C05442=1098.979,27.951,-55.035,176.233,15.027,151.969
C05443=1098.973,27.702,-55.021,176.230,15.027,151.970
C05444=1098.967,27.452,-55.005,176.228,15.026,151.970
C05445=1098.962,27.202,-54.991,176.226,15.025,151.971
C05446=1098.956,26.952,-54.976,176.224,15.025,151.971
C05447=1098.951,26.703,-54.961,176.221,15.024,151.971
C05448=1098.944,26.454,-54.946,176.219,15.023,151.972
C05449=1098.939,26.204,-54.931,176.217,15.022,151.972
C05450=1098.933,25.955,-54.916,176.215,15.022,151.972
C05451=1098.927,25.705,-54.902,176.212,15.021,151.973
C05452=1098.922,25.455,-54.887,176.210,15.020,151.973
C05453=1098.916,25.206,-54.872,176.208,15.020,151.973
C05454=1098.910,24.957,-54.857,176.206,15.019,151.974
C05455=1098.904,24.708,-54.843,176.203,15.018,151.974
C05456=1098.899,24.458,-54.828,176.201,15.018,151.974
C05457=1098.893,24.208,-54.813,176.199,15.017,151.975
C05458=1098.887,23.959,-54.799,176.197,15.016,151.975
C05459=1098.881,23.709,-54.783,176.194,15.015,151.975
C05460=1098.876,23.460,-54.769,176.192,15.015,151.976
C05461=1098.869,23.210,-54.754,176.190,15.014,151.976
C05462=1098.863,22.961,-54.740,176.188,15.013,151.976
C05463=1098.858,22.712,-54.724,176.186,15.012,151.976
C05464=1098.852,22.461,-54.710,176.183,15.012,151.977
C05465=1098.847,22.213,-54.696,176.182,15.011,151.977
C05466=1098.841,21.963,-54.680,176.180,15.010,151.977
C05467=1098.835,21.713,-54.666,176.177,15.009,151.978
C05468=1098.830,21.464,-54.652,176.175,15.009,151.978
C05469=1098.823,21.214,-54.637,176.173,15.008,151.979
C05470=1098.819,20.964,-54.622,176.171,15.008,151.979
C05471=1098.813,20.716,-54.608,176.168,15.006,151.979
C05472=1098.806,20.466,-54.593,176.166,15.006,151.979
C05473=1098.801,20.216,-54.579,176.164,15.005,151.980
C05474=1098.795,19.967,-54.564,176.162,15.005,151.980
C05475=1098.789,19.717,-54.549,176.159,15.004,151.980
C05476=1098.784,19.468,-54.535,176.157,15.003,151.981
C05477=1098.778,19.218,-54.520,176.155,15.002,151.981
C05478=1098.772,18.969,-54.505,176.153,15.002,151.981
C05479=1098.766,18.719,-54.491,176.151,15.001,151.982
C05480=1098.760,18.470,-54.477,176.149,15.000,151.982
C05481=1098.755,18.220,-54.462,176.147,14.999,151.982
C05482=1098.749,17.970,-54.447,176.145,14.999,151.983
C05483=1098.743,17.721,-54.433,176.143,14.998,151.983
C05484=1098.738,17.472,-54.419,176.140,14.997,151.983
C05485=1098.731,17.222,-54.404,176.138,14.996,151.984
C05486=1098.726,16.973,-54.390,176.136,14.996,151.984
C05487=1098.720,16.724,-54.375,176.134,14.995,151.984
C05488=1098.714,16.473,-54.361,176.131,14.994,151.985
C05489=1098.709,16.224,-54.346,176.129,14.993,151.985
C05490=1098.702,15.952,-54.331,176.127,14.993,151.985
C05491=1098.696,15.680,-54.315,176.125,14.992,151.985
C05492=1098.690,15.408,-54.300,176.123,14.991,151.986
C05493=1098.684,15.136,-54.284,176.120,14.991,151.986
C05494=1098.678,14.886,-54.269,176.118,14.989,151.986
C05495=1098.672,14.637,-54.255,176.116,14.988,151.987
C05496=1098.666,14.388,-54.241,176.114,14.988,151.987
C05497=1098.660,14.137,-54.227,176.112,14.987,151.987
C05498=1098.655,13.889,-54.212,176.109,14.986,151.988
C05499=1098.649,13.639,-54.198,176.107,14.985,151.988
C05500=1098.643,13.389,-54.183,176.105,14.985,151.988
C05501=1098.637,13.140,-54.169,176.103,14.984,151.989
C05502=1098.631,12.891,-54.155,176.101,14.984,151.989
C05503=1098.625,12.640,-54.140,176.098,14.983,151.989
C05504=1098.620,12.391,-54.127,176.097,14.982,151.990
C05505=1098.614,12.142,-54.112,176.095,14.981,151.990
C05506=1098.608,11.892,-54.098,176.092,14.981,151.990
C05507=1098.602,11.642,-54.085,176.091,14.980,151.990
C05508=1098.596,11.393,-54.070,176.088,14.979,151.991
C05509=1098.590,11.143,-54.056,176.086,14.978,151.991
C05510=1098.584,10.894,-54.041,176.084,14.978,151.991
C05511=1098.579,10.645,-54.027,176.082,14.977,151.992
C05512=1098.573,10.394,-54.013,176.080,14.976,151.992
C05513=1098.567,10.145,-53.998,176.077,14.975,151.992
C05514=1098.561,9.896,-53.985,176.075,14.975,151.993
C05515=1098.556,9.646,-53.971,176.073,14.974,151.993
C05516=1098.550,9.397,-53.956,176.072,14.973,151.993
C05517=1098.543,9.147,-53.943,176.070,14.972,151.993
C05518=1098.538,8.898,-53.929,176.067,14.972,151.994
C05519=1098.532,8.648,-53.915,176.065,14.971,151.994
C05520=1098.526,8.399,-53.900,176.063,14.970,151.994
C05521=1098.520,8.149,-53.886,176.061,14.969,151.995
C05522=1098.515,7.899,-53.872,176.059,14.969,151.995
C05523=1098.510,7.650,-53.858,176.056,14.968,151.995
C05524=1098.502,7.400,-53.844,176.054,14.967,151.996
C05525=1098.497,7.151,-53.830,176.052,14.966,151.996
C05526=1098.491,6.901,-53.816,176.051,14.965,151.996
C05527=1098.486,6.652,-53.802,176.048,14.965,151.997
C05528=1098.480,6.402,-53.787,176.046,14.964,151.997
C05529=1098.474,6.153,-53.773,176.044,14.963,151.997
C05530=1098.469,5.903,-53.760,176.042,14.962,151.997
C05531=1098.462,5.654,-53.746,176.040,14.962,151.998
C05532=1098.457,5.404,-53.732,176.038,14.961,151.998
C05533=1098.451,5.154,-53.718,176.036,14.961,151.998
C05534=1098.445,4.905,-53.704,176.033,14.959,151.999
C05535=1098.440,4.655,-53.690,176.031,14.958,151.999
C05536=1098.433,4.406,-53.677,176.030,14.958,151.999
C05537=1098.428,4.156,-53.663,176.028,14.957,151.999
C05538=1098.422,3.907,-53.649,176.026,14.956,152.000
C05539=1098.416,3.657,-53.635,176.023,14.955,152.000
C05540=1098.411,3.408,-53.620,176.021,14.955,152.000
C05541=1098.404,3.158,-53.607,176.019,14.954,152.001
C05542=1098.399,2.909,-53.593,176.017,14.953,152.001
C05543=1098.393,2.659,-53.579,176.015,14.952,152.001
C05544=1098.388,2.410,-53.565,176.014,14.952,152.001
C05545=1098.382,2.160,-53.551,176.011,14.950,152.002
C05546=1098.376,1.910,-53.538,176.009,14.950,152.002
C05547=1098.370,1.661,-53.524,176.007,14.949,152.002
C05548=1098.365,1.411,-53.510,176.005,14.949,152.003
C05549=1098.359,1.161,-53.496,176.003,14.948,152.003
C05550=1098.353,0.912,-53.483,176.001,14.947,152.003
C05551=1098.348,0.663,-53.469,175.998,14.946,152.003
C05552=1098.342,0.413,-53.455,175.997,14.945,152.004
C05553=1098.337,0.163,-53.441,175.995,14.944,152.004
C05554=1098.330,-0.107,-53.426,175.993,14.943,152.004
C05555=1098.324,-0.377,-53.412,175.990,14.942,152.004
C05556=1098.317,-0.646,-53.396,175.988,14.941,152.005
C05557=1098.311,-0.917,-53.381,175.986,14.941,152.005
C05558=1098.305,-1.166,-53.368,175.983,14.940,152.005
C05559=1098.300,-1.416,-53.354,175.982,14.939,152.006
C05560=1098.294,-1.665,-53.340,175.980,14.938,152.006
C05561=1098.289,-1.915,-53.327,175.978,14.938,152.006
C05562=1098.283,-2.165,-53.314,175.976,14.937,152.006
C05563=1098.277,-2.414,-53.300,175.974,14.936,152.007
C05564=1098.272,-2.664,-53.286,175.971,14.935,152.007
C05565=1098.265,-2.913,-53.273,175.970,14.934,152.007
C05566=1098.260,-3.163,-53.259,175.968,14.933,152.007
C05567=1098.255,-3.412,-53.245,175.966,14.932,152.008
C05568=1098.248,-3.661,-53.232,175.964,14.932,152.008
C05569=1098.242,-3.912,-53.218,175.962,14.931,152.008
C05570=1098.236,-4.161,-53.204,175.960,14.930,152.008
C05571=1098.231,-4.411,-53.190,175.957,14.929,152.009
C05572=1098.225,-4.660,-53.178,175.955,14.929,152.009
C05573=1098.219,-4.910,-53.164,175.953,14.928,152.009
C05574=1098.213,-5.159,-53.151,175.952,14.927,152.010
C05575=1098.207,-5.409,-53.137,175.950,14.926,152.010
C05576=1098.201,-5.658,-53.124,175.948,14.926,152.010
C05577=1098.196,-5.908,-53.110,175.946,14.925,152.010
C05578=1098.190,-6.157,-53.096,175.943,14.924,152.011
C05579=1098.184,-6.408,-53.083,175.941,14.923,152.011
C05580=1098.178,-6.657,-53.070,175.940,14.922,152.011
C05581=1098.172,-6.907,-53.056,175.938,14.921,152.012
C05582=1098.166,-7.156,-53.042,175.935,14.921,152.012
C05583=1098.160,-7.406,-53.029,175.934,14.920,152.012
C05584=1098.155,-7.655,-53.016,175.932,14.920,152.013
C05585=1098.149,-7.905,-53.002,175.930,14.919,152.013
C05586=1098.143,-8.154,-52.989,175.927,14.917,152.013
C05587=1098.137,-8.404,-52.975,175.925,14.917,152.013
C05588=1098.131,-8.653,-52.962,175.923,14.916,152.014
C05589=1098.126,-8.903,-52.949,175.922,14.915,152.014
C05590=1098.120,-9.153,-52.935,175.920,14.915,152.014
C05591=1098.114,-9.402,-52.922,175.918,14.914,152.014
C05592=1098.108,-9.652,-52.909,175.916,14.913,152.015
C05593=1098.102,-9.901,-52.896,175.914,14.912,152.015
C05594=1098.097,-10.151,-52.882,175.911,14.911,152.015
C05595=1098.090,-10.400,-52.869,175.909,14.910,152.015
C05596=1098.085,-10.650,-52.855,175.908,14.909,152.016
C05597=1098.079,-10.900,-52.842,175.906,14.909,152.016
C05598=1098.074,-11.149,-52.828,175.904,14.908,152.016
C05599=1098.068,-11.399,-52.816,175.902,14.907,152.016
C05600=1098.061,-11.648,-52.802,175.900,14.906,152.017
C05601=1098.056,-11.898,-52.789,175.898,14.906,152.017
C05602=1098.050,-12.148,-52.776,175.896,14.904,152.017
C05603=1098.045,-12.397,-52.762,175.894,14.904,152.018
C05604=1098.038,-12.647,-52.749,175.892,14.903,152.018
C05605=1098.033,-12.896,-52.736,175.890,14.902,152.018
C05606=1098.027,-13.146,-52.722,175.888,14.901,152.018
C05607=1098.021,-13.396,-52.710,175.886,14.901,152.019
C05608=1098.016,-13.645,-52.696,175.884,14.900,152.019
C05609=1098.009,-13.895,-52.683,175.882,14.899,152.019
C05610=1098.004,-14.144,-52.671,175.881,14.898,152.019
C05611=1097.999,-14.393,-52.657,175.878,14.897,152.020
C05612=1097.993,-14.643,-52.644,175.876,14.896,152.020
C05613=1097.987,-14.893,-52.631,175.874,14.896,152.020
C05614=1097.981,-15.143,-52.618,175.872,14.895,152.020
C05615=1097.975,-15.392,-52.605,175.870,14.894,152.021
C05616=1097.969,-15.641,-52.591,175.868,14.893,152.021
C05617=1097.963,-15.891,-52.579,175.867,14.893,152.021
C05618=1097.957,-16.160,-52.564,175.865,14.892,152.021
C05619=1097.950,-16.428,-52.551,175.862,14.891,152.022
C05620=1097.944,-16.697,-52.536,175.860,14.890,152.022
C05621=1097.938,-16.965,-52.523,175.858,14.890,152.022
C05622=1097.932,-17.214,-52.509,175.856,14.889,152.023
C05623=1097.927,-17.465,-52.496,175.854,14.888,152.023
C05624=1097.920,-17.714,-52.483,175.852,14.887,152.023
C05625=1097.914,-17.964,-52.470,175.850,14.886,152.023
C05626=1097.908,-18.213,-52.457,175.848,14.885,152.024
C05627=1097.902,-18.463,-52.444,175.846,14.885,152.024
C05628=1097.897,-18.712,-52.431,175.844,14.884,152.024
C05629=1097.892,-18.962,-52.418,175.842,14.883,152.025
C05630=1097.885,-19.211,-52.405,175.840,14.882,152.025
C05631=1097.879,-19.461,-52.393,175.838,14.882,152.025
C05632=1097.873,-19.710,-52.379,175.837,14.881,152.025
C05633=1097.867,-19.960,-52.367,175.835,14.880,152.026
C05634=1097.862,-20.210,-52.354,175.833,14.879,152.026
C05635=1097.856,-20.459,-52.340,175.831,14.879,152.026
C05636=1097.850,-20.709,-52.328,175.829,14.878,152.026
C05637=1097.844,-20.959,-52.315,175.827,14.877,152.026
C05638=1097.839,-21.208,-52.302,175.825,14.875,152.027
C05639=1097.833,-21.458,-52.290,175.823,14.875,152.027
C05640=1097.827,-21.707,-52.276,175.821,14.874,152.027
C05641=1097.821,-21.957,-52.263,175.819,14.873,152.027
C05642=1097.815,-22.206,-52.250,175.817,14.872,152.028
C05643=1097.809,-22.456,-52.238,175.815,14.872,152.028
C05644=1097.803,-22.706,-52.225,175.814,14.871,152.028
C05645=1097.798,-22.955,-52.212,175.812,14.870,152.029
C05646=1097.792,-23.205,-52.200,175.810,14.869,152.029
C05647=1097.786,-23.455,-52.187,175.808,14.869,152.029
C05648=1097.780,-23.704,-52.173,175.806,14.868,152.029
C05649=1097.774,-23.954,-52.161,175.804,14.867,152.030
C05650=1097.768,-24.204,-52.148,175.802,14.866,152.030
C05651=1097.763,-24.453,-52.136,175.800,14.866,152.030
C05652=1097.757,-24.702,-52.123,175.798,14.864,152.030
C05653=1097.751,-24.952,-52.110,175.796,14.864,152.031
C05654=1097.745,-25.202,-52.097,175.794,14.863,152.031
C05655=1097.739,-25.451,-52.084,175.792,14.862,152.031
C05656=1097.734,-25.701,-52.072,175.790,14.861,152.031
C05657=1097.728,-25.951,-52.059,175.789,14.860,152.032
C05658=1097.723,-26.201,-52.046,175.787,14.859,152.032
C05659=1097.717,-26.450,-52.034,175.785,14.859,152.032
C05660=1097.710,-26.700,-52.020,175.783,14.858,152.032
C05661=1097.705,-26.949,-52.008,175.781,14.857,152.033
C05662=1097.699,-27.199,-51.996,175.779,14.857,152.033
C05663=1097.693,-27.449,-51.983,175.777,14.856,152.033
C05664=1097.687,-27.698,-51.970,175.776,14.855,152.033
C05665=1097.681,-27.948,-51.957,175.774,14.854,152.034
C05666=1097.676,-28.197,-51.945,175.772,14.854,152.034
C05667=1097.669,-28.447,-51.933,175.770,14.853,152.034
C05668=1097.663,-28.696,-51.921,175.768,14.852,152.034
C05669=1097.657,-28.946,-51.907,175.766,14.851,152.035
C05670=1097.651,-29.196,-51.895,175.764,14.851,152.035
C05671=1097.646,-29.445,-51.883,175.762,14.850,152.035
C05672=1097.640,-29.695,-51.870,175.760,14.849,152.035
C05673=1097.634,-29.945,-51.858,175.759,14.848,152.036
C05674=1097.628,-30.194,-51.845,175.757,14.848,152.036
C05675=1097.622,-30.444,-51.832,175.754,14.846,152.036
C05676=1097.617,-30.693,-51.819,175.752,14.846,152.036
C05677=1097.611,-30.943,-51.807,175.750,14.845,152.037
C05678=1097.604,-31.192,-51.795,175.748,14.844,152.037
C05679=1097.598,-31.442,-51.782,175.747,14.843,152.037
C05680=1097.593,-31.691,-51.770,175.745,14.842,152.037
C05681=1097.587,-31.941,-51.758,175.743,14.841,152.038
C05682=1097.581,-32.209,-51.744,175.741,14.841,152.038
C05683=1097.575,-32.477,-51.731,175.739,14.840,152.038
C05684=1097.567,-32.744,-51.717,175.737,14.839,152.038
C05685=1097.561,-33.012,-51.704,175.736,14.839,152.039
C05686=1097.556,-33.261,-51.692,175.734,14.838,152.039
C05687=1097.550,-33.511,-51.680,175.732,14.837,152.039
C05688=1097.544,-33.761,-51.667,175.730,14.836,152.039
C05689=1097.538,-34.010,-51.654,175.728,14.836,152.040
C05690=1097.532,-34.259,-51.642,175.726,14.835,152.040
C05691=1097.526,-34.509,-51.630,175.724,14.834,152.040
C05692=1097.520,-34.759,-51.617,175.722,14.833,152.040
C05693=1097.515,-35.008,-51.605,175.721,14.833,152.041
C05694=1097.509,-35.258,-51.592,175.719,14.832,152.041
C05695=1097.503,-35.508,-51.580,175.717,14.831,152.041
C05696=1097.497,-35.758,-51.569,175.715,14.830,152.042
C05697=1097.492,-36.007,-51.556,175.713,14.830,152.042
C05698=1097.486,-36.257,-51.544,175.711,14.829,152.042
C05699=1097.480,-36.507,-51.531,175.709,14.827,152.042
C05700=1097.474,-36.756,-51.519,175.707,14.826,152.042
C05701=1097.468,-37.006,-51.507,175.705,14.826,152.043
C05702=1097.462,-37.256,-51.495,175.703,14.825,152.043
C05703=1097.457,-37.505,-51.482,175.701,14.824,152.043
C05704=1097.451,-37.755,-51.470,175.699,14.823,152.044
C05705=1097.445,-38.005,-51.457,175.698,14.823,152.044
C05706=1097.439,-38.254,-51.445,175.696,14.822,152.044
C05707=1097.433,-38.503,-51.433,175.695,14.822,152.044
C05708=1097.427,-38.753,-51.421,175.693,14.821,152.044
C05709=1097.422,-39.003,-51.408,175.691,14.820,152.045
C05710=1097.415,-39.253,-51.397,175.689,14.819,152.045
C05711=1097.409,-39.503,-51.385,175.687,14.818,152.045
C05712=1097.404,-39.752,-51.372,175.685,14.818,152.045
C05713=1097.397,-40.001,-51.360,175.684,14.817,152.046
C05714=1097.391,-40.251,-51.348,175.682,14.816,152.046
C05715=1097.386,-40.500,-51.336,175.680,14.816,152.046
C05716=1097.379,-40.750,-51.324,175.678,14.815,152.046
C05717=1097.374,-41.000,-51.312,175.676,14.814,152.047
C05718=1097.369,-41.250,-51.300,175.674,14.813,152.047
C05719=1097.362,-41.499,-51.288,175.672,14.813,152.047
C05720=1097.356,-41.749,-51.275,175.670,14.812,152.047
C05721=1097.350,-41.998,-51.264,175.669,14.811,152.048
C05722=1097.344,-42.248,-51.251,175.667,14.810,152.048
C05723=1097.338,-42.498,-51.239,175.665,14.810,152.048
C05724=1097.332,-42.747,-51.228,175.663,14.809,152.049
C05725=1097.326,-42.997,-51.215,175.661,14.808,152.049
C05726=1097.321,-43.247,-51.203,175.659,14.807,152.049
C05727=1097.315,-43.497,-51.192,175.657,14.807,152.049
C05728=1097.309,-43.746,-51.179,175.656,14.806,152.049
C05729=1097.303,-43.995,-51.168,175.654,14.805,152.050
C05730=1097.297,-44.245,-51.155,175.652,14.804,152.050
C05731=1097.291,-44.496,-51.143,175.650,14.803,152.050
C05732=1097.285,-44.745,-51.132,175.648,14.803,152.050
C05733=1097.279,-44.994,-51.119,175.646,14.802,152.051
C05734=1097.273,-45.243,-51.107,175.644,14.801,152.051
C05735=1097.268,-45.494,-51.096,175.643,14.800,152.051
C05736=1097.261,-45.743,-51.084,175.641,14.800,152.052
C05737=1097.256,-45.993,-51.071,175.639,14.799,152.052
C05738=1097.250,-46.243,-51.060,175.637,14.798,152.052
C05739=1097.244,-46.492,-51.048,175.635,14.797,152.052
C05740=1097.238,-46.742,-51.035,175.634,14.797,152.053
C05741=1097.232,-46.992,-51.024,175.632,14.797,152.053
C05742=1097.227,-47.241,-51.012,175.630,14.795,152.053
C05743=1097.220,-47.491,-51.000,175.629,14.795,152.053
C05744=1097.215,-47.741,-50.989,175.627,14.794,152.053
C05745=1097.208,-47.990,-50.977,175.625,14.793,152.054
C05746=1097.202,-48.258,-50.964,175.623,14.792,152.054
C05747=1097.196,-48.526,-50.951,175.621,14.792,152.054
C05748=1097.190,-48.794,-50.938,175.619,14.791,152.054
C05749=1097.183,-49.061,-50.926,175.616,14.790,152.055
C05750=1097.178,-49.312,-50.914,175.615,14.790,152.055
C05751=1097.172,-49.561,-50.902,175.614,14.789,152.055
C05752=1097.166,-49.810,-50.890,175.612,14.788,152.055
C05753=1097.160,-50.060,-50.879,175.610,14.787,152.056
C05754=1097.154,-50.310,-50.866,175.608,14.787,152.056
C05755=1097.148,-50.559,-50.855,175.606,14.786,152.056
C05756=1097.142,-50.809,-50.843,175.604,14.785,152.057
C05757=1097.136,-51.059,-50.832,175.602,14.784,152.057
C05758=1097.130,-51.308,-50.820,175.600,14.784,152.057
C05759=1097.124,-51.558,-50.807,175.598,14.783,152.057
C05760=1097.118,-51.808,-50.797,175.597,14.782,152.058
C05761=1097.112,-52.057,-50.785,175.595,14.782,152.058
C05762=1097.106,-52.308,-50.773,175.593,14.781,152.058
C05763=1097.100,-52.557,-50.761,175.592,14.781,152.058
C05764=1097.094,-52.807,-50.750,175.590,14.780,152.059
C05765=1097.089,-53.056,-50.738,175.588,14.779,152.059
C05766=1097.082,-53.306,-50.727,175.586,14.778,152.059
C05767=1097.076,-53.555,-50.715,175.584,14.778,152.059
C05768=1097.070,-53.805,-50.704,175.582,14.777,152.060
C05769=1097.064,-54.055,-50.691,175.580,14.776,152.060
C05770=1097.058,-54.305,-50.680,175.579,14.776,152.060
C05771=1097.051,-54.554,-50.668,175.577,14.775,152.060
C05772=1097.046,-54.804,-50.657,175.575,14.774,152.061
C05773=1097.040,-55.054,-50.645,175.573,14.773,152.061
C05774=1097.034,-55.303,-50.634,175.572,14.773,152.061
C05775=1097.027,-55.553,-50.622,175.570,14.773,152.061
C05776=1097.022,-55.802,-50.611,175.568,14.772,152.062
C05777=1097.016,-56.052,-50.599,175.566,14.771,152.062
C05778=1097.010,-56.301,-50.588,175.564,14.770,152.062
C05779=1097.004,-56.552,-50.576,175.562,14.770,152.063
C05780=1096.998,-56.801,-50.565,175.561,14.769,152.063
C05781=1096.992,-57.051,-50.553,175.559,14.768,152.063
C05782=1096.986,-57.300,-50.541,175.557,14.767,152.063
C05783=1096.980,-57.550,-50.530,175.556,14.767,152.064
C05784=1096.974,-57.799,-50.519,175.554,14.767,152.064
C05785=1096.968,-58.049,-50.507,175.552,14.766,152.064
C05786=1096.962,-58.299,-50.496,175.550,14.765,152.064
C05787=1096.956,-58.549,-50.484,175.548,14.764,152.064
C05788=1096.950,-58.798,-50.473,175.547,14.763,152.065
C05789=1096.944,-59.048,-50.462,175.545,14.762,152.065
C05790=1096.938,-59.297,-50.450,175.543,14.762,152.065
C05791=1096.932,-59.548,-50.438,175.542,14.762,152.065
C05792=1096.926,-59.797,-50.427,175.540,14.761,152.066
C05793=1096.920,-60.047,-50.416,175.538,14.760,152.066
C05794=1096.914,-60.296,-50.405,175.536,14.759,152.066
C05795=1096.908,-60.547,-50.393,175.534,14.759,152.066
C05796=1096.902,-60.796,-50.381,175.532,14.758,152.067
C05797=1096.896,-61.046,-50.370,175.530,14.757,152.067
C05798=1096.890,-61.295,-50.359,175.529,14.757,152.067
C05799=1096.884,-61.544,-50.348,175.527,14.756,152.068
C05800=1096.878,-61.794,-50.336,175.526,14.756,152.068
C05801=1096.873,-62.044,-50.325,175.524,14.755,152.068
C05802=1096.866,-62.294,-50.314,175.522,14.754,152.068
C05803=1096.860,-62.543,-50.302,175.520,14.753,152.069
C05804=1096.855,-62.793,-50.291,175.518,14.753,152.069
C05805=1096.848,-63.043,-50.280,175.516,14.752,152.069
C05806=1096.842,-63.292,-50.269,175.515,14.752,152.069
C05807=1096.837,-63.542,-50.256,175.513,14.751,152.070
C05808=1096.831,-63.792,-50.246,175.511,14.750,152.070
C05809=1096.825,-64.042,-50.234,175.509,14.750,152.070
C05810=1096.818,-64.310,-50.223,175.507,14.749,152.070
C05811=1096.812,-64.579,-50.210,175.506,14.748,152.071
C05812=1096.805,-64.849,-50.199,175.504,14.748,152.071
C05813=1096.799,-65.118,-50.186,175.502,14.747,152.071
C05814=1096.793,-65.368,-50.175,175.500,14.746,152.071
C05815=1096.787,-65.618,-50.164,175.498,14.745,152.072
C05816=1096.781,-65.867,-50.152,175.496,14.745,152.072
C05817=1096.775,-66.117,-50.141,175.495,14.745,152.072
C05818=1096.770,-66.367,-50.129,175.493,14.744,152.072
C05819=1096.764,-66.616,-50.119,175.491,14.743,152.073
C05820=1096.758,-66.866,-50.107,175.489,14.742,152.073
C05821=1096.752,-67.116,-50.096,175.488,14.742,152.073
C05822=1096.746,-67.365,-50.086,175.486,14.741,152.074
C05823=1096.740,-67.615,-50.074,175.485,14.741,152.074
C05824=1096.734,-67.865,-50.063,175.483,14.740,152.074
C05825=1096.728,-68.114,-50.052,175.481,14.739,152.074
C05826=1096.722,-68.364,-50.041,175.479,14.739,152.075
C05827=1096.716,-68.614,-50.030,175.477,14.738,152.075
C05828=1096.710,-68.863,-50.019,175.475,14.737,152.075
C05829=1096.705,-69.114,-50.007,175.474,14.737,152.075
C05830=1096.699,-69.363,-49.996,175.472,14.736,152.076
C05831=1096.693,-69.613,-49.985,175.470,14.736,152.076
C05832=1096.687,-69.863,-49.974,175.468,14.735,152.076
C05833=1096.681,-70.112,-49.962,175.467,14.734,152.076
C05834=1096.675,-70.361,-49.952,175.465,14.733,152.077
C05835=1096.669,-70.611,-49.941,175.464,14.733,152.077
C05836=1096.663,-70.861,-49.929,175.462,14.733,152.077
C05837=1096.657,-71.110,-49.919,175.460,14.732,152.077
C05838=1096.652,-71.360,-49.908,175.458,14.731,152.078
C05839=1096.645,-71.610,-49.896,175.456,14.730,152.078
C05840=1096.639,-71.860,-49.886,175.455,14.730,152.078
C05841=1096.634,-72.109,-49.875,175.453,14.730,152.078
C05842=1096.628,-72.359,-49.864,175.451,14.729,152.079
C05843=1096.622,-72.609,-49.853,175.450,14.728,152.079
C05844=1096.616,-72.858,-49.842,175.448,14.727,152.079
C05845=1096.610,-73.108,-49.831,175.446,14.726,152.079
C05846=1096.604,-73.357,-49.820,175.445,14.726,152.079
C05847=1096.599,-73.608,-49.808,175.443,14.725,152.080
C05848=1096.593,-73.857,-49.797,175.441,14.725,152.080
C05849=1096.587,-74.107,-49.786,175.439,14.724,152.080
C05850=1096.581,-74.356,-49.776,175.437,14.723,152.081
C05851=1096.575,-74.606,-49.765,175.436,14.723,152.081
C05852=1096.569,-74.856,-49.754,175.434,14.722,152.081
C05853=1096.563,-75.106,-49.744,175.432,14.722,152.081
C05854=1096.557,-75.356,-49.733,175.430,14.721,152.082
C05855=1096.551,-75.605,-49.722,175.429,14.721,152.082
C05856=1096.546,-75.855,-49.711,175.427,14.720,152.082
C05857=1096.539,-76.105,-49.700,175.425,14.720,152.082
C05858=1096.533,-76.354,-49.689,175.423,14.719,152.083
C05859=1096.527,-76.604,-49.678,175.421,14.718,152.083
C05860=1096.521,-76.853,-49.667,175.420,14.718,152.083
C05861=1096.515,-77.103,-49.656,175.418,14.717,152.084
C05862=1096.509,-77.353,-49.645,175.417,14.717,152.084
C05863=1096.503,-77.602,-49.634,175.415,14.716,152.084
C05864=1096.497,-77.851,-49.624,175.414,14.716,152.084
C05865=1096.491,-78.102,-49.614,175.412,14.715,152.085
C05866=1096.485,-78.352,-49.603,175.410,14.714,152.085
C05867=1096.479,-78.601,-49.592,175.408,14.714,152.085
C05868=1096.474,-78.851,-49.581,175.406,14.713,152.085
C05869=1096.467,-79.101,-49.570,175.405,14.713,152.086
C05870=1096.461,-79.350,-49.560,175.403,14.712,152.086
C05871=1096.455,-79.600,-49.549,175.401,14.712,152.086
C05872=1096.450,-79.850,-49.538,175.399,14.711,152.087
C05873=1096.443,-80.100,-49.527,175.398,14.711,152.087
C05874=1096.436,-80.371,-49.516,175.396,14.710,152.087
C05875=1096.430,-80.642,-49.505,175.394,14.710,152.087
C05876=1096.424,-80.914,-49.493,175.392,14.709,152.088
C05877=1096.417,-81.185,-49.482,175.390,14.709,152.088
C05878=1096.411,-81.434,-49.471,175.388,14.708,152.088
C05879=1096.405,-81.685,-49.459,175.387,14.708,152.088
C05880=1096.398,-81.934,-49.449,175.385,14.707,152.089
C05881=1096.393,-82.184,-49.439,175.383,14.706,152.089
C05882=1096.387,-82.433,-49.428,175.381,14.706,152.089
C05883=1096.380,-82.683,-49.418,175.380,14.706,152.089
C05884=1096.374,-82.933,-49.407,175.378,14.705,152.090
C05885=1096.369,-83.183,-49.396,175.376,14.705,152.090
C05886=1096.362,-83.432,-49.386,175.374,14.704,152.090
C05887=1096.356,-83.682,-49.375,175.373,14.704,152.091
C05888=1096.350,-83.932,-49.364,175.371,14.703,152.091
C05889=1096.344,-84.182,-49.355,175.369,14.702,152.091
C05890=1096.338,-84.431,-49.344,175.368,14.702,152.091
C05891=1096.331,-84.681,-49.333,175.366,14.702,152.092
C05892=1096.325,-84.930,-49.322,175.364,14.701,152.092
C05893=1096.320,-85.181,-49.312,175.362,14.701,152.092
C05894=1096.313,-85.430,-49.302,175.361,14.700,152.093
C05895=1096.308,-85.679,-49.291,175.359,14.700,152.093
C05896=1096.301,-85.930,-49.281,175.357,14.699,152.093
C05897=1096.295,-86.179,-49.270,175.356,14.698,152.093
C05898=1096.289,-86.429,-49.259,175.354,14.699,152.094
C05899=1096.283,-86.679,-49.250,175.352,14.698,152.094
C05900=1096.278,-86.928,-49.239,175.350,14.697,152.094
C05901=1096.270,-87.178,-49.228,175.348,14.696,152.095
C05902=1096.265,-87.428,-49.218,175.347,14.696,152.095
C05903=1096.259,-87.677,-49.207,175.346,14.696,152.095
C05904=1096.253,-87.927,-49.197,175.344,14.695,152.095
C05905=1096.247,-88.177,-49.187,175.342,14.695,152.096
C05906=1096.240,-88.427,-49.176,175.340,14.695,152.096
C05907=1096.235,-88.676,-49.165,175.338,14.694,152.096
C05908=1096.228,-88.926,-49.155,175.337,14.694,152.097
C05909=1096.223,-89.175,-49.145,175.335,14.693,152.097
C05910=1096.217,-89.426,-49.134,175.334,14.692,152.097
C05911=1096.211,-89.675,-49.124,175.332,14.692,152.097
C05912=1096.205,-89.924,-49.113,175.330,14.692,152.098
C05913=1096.198,-90.175,-49.103,175.328,14.691,152.098
C05914=1096.193,-90.424,-49.092,175.326,14.691,152.098
C05915=1096.186,-90.674,-49.083,175.325,14.690,152.098
C05916=1096.181,-90.923,-49.072,175.323,14.690,152.099
C05917=1096.174,-91.173,-49.062,175.322,14.689,152.099
C05918=1096.169,-91.423,-49.052,175.320,14.689,152.099
C05919=1096.162,-91.672,-49.041,175.318,14.689,152.100
C05920=1096.157,-91.922,-49.031,175.316,14.688,152.100
C05921=1096.150,-92.172,-49.020,175.315,14.687,152.100
C05922=1096.144,-92.422,-49.010,175.313,14.687,152.100
C05923=1096.139,-92.672,-48.999,175.312,14.686,152.101
C05924=1096.132,-92.921,-48.990,175.309,14.686,152.101
C05925=1096.127,-93.171,-48.979,175.308,14.686,152.101
C05926=1096.120,-93.421,-48.969,175.306,14.685,152.102
C05927=1096.115,-93.670,-48.959,175.304,14.685,152.102
C05928=1096.109,-93.920,-48.949,175.303,14.684,152.102
C05929=1096.103,-94.169,-48.938,175.301,14.684,152.102
C05930=1096.097,-94.419,-48.928,175.299,14.684,152.103
C05931=1096.091,-94.669,-48.918,175.298,14.683,152.103
C05932=1096.084,-94.919,-48.908,175.296,14.683,152.103
C05933=1096.079,-95.169,-48.898,175.294,14.682,152.104
C05934=1096.072,-95.418,-48.887,175.293,14.682,152.104
C05935=1096.067,-95.669,-48.877,175.291,14.681,152.104
C05936=1096.060,-95.918,-48.867,175.289,14.681,152.104
C05937=1096.055,-96.168,-48.857,175.288,14.681,152.105
C05938=1096.048,-96.441,-48.845,175.286,14.680,152.105
C05939=1096.042,-96.714,-48.834,175.284,14.679,152.105
C05940=1096.035,-96.988,-48.824,175.282,14.679,152.106
C05941=1096.028,-97.262,-48.813,175.280,14.678,152.106
C05942=1096.022,-97.512,-48.802,175.279,14.678,152.106
C05943=1096.016,-97.762,-48.792,175.277,14.678,152.106
C05944=1096.011,-98.012,-48.782,175.275,14.677,152.107
C05945=1096.004,-98.261,-48.772,175.274,14.677,152.107
C05946=1095.998,-98.511,-48.762,175.272,14.677,152.107
C05947=1095.992,-98.761,-48.751,175.270,14.676,152.108
C05948=1095.986,-99.011,-48.741,175.269,14.676,152.108
C05949=1095.980,-99.260,-48.732,175.267,14.675,152.108
C05950=1095.974,-99.510,-48.721,175.266,14.675,152.109
C05951=1095.968,-99.760,-48.711,175.263,14.675,152.109
C05952=1095.961,-100.009,-48.702,175.262,14.674,152.109
C05953=1095.955,-100.259,-48.692,175.260,14.674,152.109
C05954=1095.950,-100.509,-48.681,175.259,14.674,152.110
C05955=1095.943,-100.759,-48.672,175.256,14.673,152.110
C05956=1095.937,-101.008,-48.661,175.255,14.673,152.110
C05957=1095.931,-101.258,-48.651,175.253,14.673,152.111
C05958=1095.925,-101.508,-48.642,175.252,14.672,152.111
C05959=1095.919,-101.757,-48.631,175.250,14.672,152.111
C05960=1095.913,-102.007,-48.621,175.248,14.671,152.112
C05961=1095.907,-102.257,-48.612,175.247,14.671,152.112
C05962=1095.901,-102.506,-48.601,175.245,14.671,152.112
C05963=1095.895,-102.756,-48.592,175.243,14.670,152.112
C05964=1095.889,-103.006,-48.582,175.242,14.670,152.113
C05965=1095.883,-103.255,-48.571,175.240,14.670,152.113
C05966=1095.876,-103.505,-48.562,175.239,14.670,152.113
C05967=1095.870,-103.755,-48.552,175.237,14.669,152.114
C05968=1095.864,-104.005,-48.542,175.235,14.669,152.114
C05969=1095.858,-104.255,-48.532,175.233,14.669,152.114
C05970=1095.852,-104.504,-48.522,175.232,14.668,152.115
C05971=1095.845,-104.754,-48.512,175.230,14.668,152.115
C05972=1095.840,-105.004,-48.502,175.229,14.667,152.115
C05973=1095.834,-105.253,-48.492,175.226,14.667,152.115
C05974=1095.827,-105.503,-48.482,175.225,14.667,152.116
C05975=1095.821,-105.753,-48.473,175.223,14.666,152.116
C05976=1095.816,-106.003,-48.463,175.221,14.666,152.116
C05977=1095.810,-106.253,-48.453,175.220,14.666,152.117
C05978=1095.803,-106.502,-48.443,175.218,14.665,152.117
C05979=1095.797,-106.752,-48.433,175.217,14.666,152.117
C05980=1095.791,-107.002,-48.424,175.215,14.665,152.118
C05981=1095.785,-107.251,-48.414,175.213,14.664,152.118
C05982=1095.780,-107.501,-48.404,175.211,14.665,152.118
C05983=1095.773,-107.750,-48.394,175.210,14.664,152.118
C05984=1095.767,-108.000,-48.384,175.208,14.664,152.119
C05985=1095.761,-108.250,-48.375,175.206,14.664,152.119
C05986=1095.755,-108.500,-48.365,175.205,14.663,152.119
C05987=1095.749,-108.749,-48.356,175.203,14.663,152.120
C05988=1095.742,-108.999,-48.346,175.201,14.663,152.120
C05989=1095.737,-109.249,-48.335,175.200,14.662,152.120
C05990=1095.731,-109.498,-48.326,175.198,14.662,152.121
C05991=1095.724,-109.748,-48.316,175.197,14.662,152.121
C05992=1095.718,-109.998,-48.307,175.195,14.661,152.121
C05993=1095.712,-110.248,-48.297,175.193,14.661,152.122
C05994=1095.706,-110.498,-48.287,175.191,14.661,152.122
C05995=1095.700,-110.747,-48.278,175.190,14.660,152.122
C05996=1095.693,-110.997,-48.268,175.188,14.661,152.123
C05997=1095.687,-111.247,-48.259,175.186,14.660,152.123
C05998=1095.681,-111.496,-48.248,175.185,14.660,152.123
C05999=1095.675,-111.746,-48.239,175.183,14.660,152.123
C06000=1095.668,-111.996,-48.229,175.181,14.659,152.124
C06001=1095.663,-112.246,-48.219,175.180,14.659,152.124
C06002=1095.656,-112.509,-48.209,175.178,14.659,152.124
C06003=1095.650,-112.774,-48.199,175.176,14.659,152.125
C06004=1095.643,-113.037,-48.189,175.174,14.658,152.125
C06005=1095.637,-113.301,-48.179,175.173,14.658,152.125
C06006=1095.631,-113.550,-48.169,175.171,14.658,152.126
C06007=1095.625,-113.800,-48.160,175.169,14.657,152.126
C06008=1095.619,-114.050,-48.150,175.168,14.658,152.126
C06009=1095.613,-114.300,-48.141,175.166,14.657,152.127
C06010=1095.606,-114.550,-48.131,175.165,14.657,152.127
C06011=1095.600,-114.799,-48.121,175.163,14.657,152.127
C06012=1095.595,-115.049,-48.112,175.161,14.656,152.128
C06013=1095.588,-115.298,-48.103,175.159,14.656,152.128
C06014=1095.582,-115.548,-48.093,175.157,14.656,152.128
C06015=1095.576,-115.798,-48.083,175.156,14.656,152.129
C06016=1095.570,-116.048,-48.074,175.154,14.655,152.129
C06017=1095.564,-116.298,-48.064,175.153,14.655,152.129
C06018=1095.558,-116.547,-48.055,175.151,14.655,152.130
C06019=1095.551,-116.797,-48.045,175.150,14.655,152.130
C06020=1095.545,-117.047,-48.036,175.147,14.655,152.130
C06021=1095.539,-117.297,-48.026,175.146,14.654,152.130
C06022=1095.533,-117.546,-48.017,175.144,14.654,152.131
C06023=1095.526,-117.796,-48.008,175.143,14.654,152.131
C06024=1095.520,-118.045,-47.998,175.141,14.654,152.132
C06025=1095.514,-118.295,-47.989,175.139,14.653,152.132
C06026=1095.508,-118.545,-47.979,175.137,14.654,152.132
C06027=1095.502,-118.794,-47.970,175.136,14.653,152.132
C06028=1095.496,-119.044,-47.960,175.134,14.653,152.133
C06029=1095.490,-119.294,-47.951,175.132,14.653,152.133
C06030=1095.483,-119.544,-47.941,175.131,14.652,152.133
C06031=1095.477,-119.794,-47.931,175.129,14.652,152.134
C06032=1095.471,-120.044,-47.923,175.128,14.652,152.134
C06033=1095.465,-120.294,-47.913,175.126,14.652,152.134
C06034=1095.459,-120.543,-47.904,175.125,14.652,152.135
C06035=1095.453,-120.792,-47.895,175.122,14.652,152.135
C06036=1095.447,-121.042,-47.885,175.121,14.651,152.135
C06037=1095.440,-121.292,-47.876,175.119,14.651,152.136
C06038=1095.434,-121.542,-47.866,175.118,14.651,152.136
C06039=1095.428,-121.792,-47.857,175.116,14.651,152.136
C06040=1095.422,-122.042,-47.848,175.115,14.651,152.137
C06041=1095.416,-122.292,-47.838,175.112,14.651,152.137
C06042=1095.410,-122.541,-47.829,175.111,14.651,152.137
C06043=1095.404,-122.790,-47.820,175.109,14.650,152.138
C06044=1095.397,-123.040,-47.810,175.108,14.650,152.138
C06045=1095.391,-123.290,-47.801,175.106,14.650,152.138
C06046=1095.385,-123.540,-47.792,175.105,14.650,152.139
C06047=1095.379,-123.790,-47.782,175.102,14.650,152.139
C06048=1095.374,-124.039,-47.773,175.101,14.650,152.139
C06049=1095.367,-124.289,-47.764,175.099,14.649,152.140
C06050=1095.361,-124.539,-47.755,175.098,14.649,152.140
C06051=1095.354,-124.788,-47.745,175.096,14.649,152.140
C06052=1095.348,-125.039,-47.736,175.095,14.649,152.141
C06053=1095.342,-125.289,-47.727,175.092,14.649,152.141
C06054=1095.335,-125.538,-47.718,175.091,14.649,152.141
C06055=1095.330,-125.787,-47.708,175.089,14.648,152.142
C06056=1095.324,-126.038,-47.700,175.088,14.649,152.142
C06057=1095.318,-126.287,-47.690,175.086,14.648,152.142
C06058=1095.311,-126.537,-47.681,175.084,14.648,152.143
C06059=1095.305,-126.787,-47.672,175.083,14.648,152.143
C06060=1095.299,-127.037,-47.662,175.081,14.648,152.143
C06061=1095.293,-127.286,-47.654,175.079,14.648,152.144
C06062=1095.286,-127.548,-47.644,175.078,14.648,152.144
C06063=1095.279,-127.809,-47.635,175.076,14.648,152.145
C06064=1095.273,-128.070,-47.624,175.074,14.648,152.145
C06065=1095.273,-128.332,-47.613,175.073,14.646,152.145
C06066=1094.865,-128.352,-47.724,175.028,14.753,152.175
C06067=1094.864,-128.093,-47.736,175.029,14.755,152.175
C06068=1094.871,-127.831,-47.745,175.031,14.756,152.175
C06069=1094.877,-127.570,-47.754,175.033,14.755,152.175
C06070=1094.883,-127.309,-47.764,175.034,14.756,152.174
C06071=1094.890,-127.059,-47.773,175.036,14.756,152.174
C06072=1094.896,-126.809,-47.783,175.038,14.756,152.174
C06073=1094.902,-126.559,-47.792,175.039,14.756,152.173
C06074=1094.908,-126.310,-47.801,175.041,14.756,152.173
C06075=1094.915,-126.060,-47.810,175.043,14.756,152.173
C06076=1094.921,-125.810,-47.819,175.045,14.757,152.172
C06077=1094.927,-125.561,-47.829,175.046,14.757,152.172
C06078=1094.933,-125.311,-47.838,175.048,14.757,152.172
C06079=1094.940,-125.061,-47.847,175.049,14.757,152.171
C06080=1094.946,-124.811,-47.856,175.051,14.757,152.171
C06081=1094.951,-124.562,-47.865,175.052,14.757,152.171
C06082=1094.958,-124.312,-47.875,175.055,14.758,152.170
C06083=1094.964,-124.062,-47.885,175.056,14.758,152.170
C06084=1094.970,-123.812,-47.893,175.058,14.758,152.170
C06085=1094.977,-123.562,-47.902,175.059,14.758,152.169
C06086=1094.983,-123.313,-47.912,175.061,14.758,152.169
C06087=1094.988,-123.063,-47.921,175.062,14.758,152.169
C06088=1094.994,-122.814,-47.931,175.064,14.759,152.169
C06089=1095.001,-122.564,-47.940,175.066,14.759,152.168
C06090=1095.007,-122.314,-47.949,175.068,14.759,152.168
C06091=1095.013,-122.064,-47.958,175.069,14.759,152.167
C06092=1095.020,-121.814,-47.968,175.071,14.760,152.167
C06093=1095.026,-121.564,-47.977,175.072,14.759,152.167
C06094=1095.032,-121.315,-47.987,175.074,14.760,152.167
C06095=1095.037,-121.065,-47.996,175.076,14.759,152.166
C06096=1095.044,-120.816,-48.006,175.078,14.760,152.166
C06097=1095.050,-120.565,-48.014,175.079,14.760,152.166
C06098=1095.056,-120.316,-48.023,175.081,14.760,152.165
C06099=1095.063,-120.066,-48.033,175.082,14.761,152.165
C06100=1095.069,-119.816,-48.043,175.084,14.761,152.165
C06101=1095.075,-119.566,-48.052,175.085,14.761,152.164
C06102=1095.081,-119.317,-48.062,175.088,14.761,152.164
C06103=1095.087,-119.067,-48.071,175.089,14.762,152.164
C06104=1095.093,-118.818,-48.080,175.091,14.761,152.163
C06105=1095.099,-118.568,-48.090,175.093,14.762,152.163
C06106=1095.105,-118.318,-48.100,175.094,14.762,152.163
C06107=1095.111,-118.068,-48.109,175.096,14.762,152.162
C06108=1095.118,-117.819,-48.119,175.097,14.763,152.162
C06109=1095.123,-117.568,-48.128,175.099,14.763,152.162
C06110=1095.130,-117.319,-48.137,175.100,14.763,152.161
C06111=1095.136,-117.069,-48.146,175.102,14.764,152.161
C06112=1095.143,-116.819,-48.156,175.104,14.763,152.161
C06113=1095.148,-116.570,-48.165,175.106,14.764,152.161
C06114=1095.154,-116.320,-48.174,175.107,14.764,152.160
C06115=1095.161,-116.070,-48.184,175.109,14.764,152.160
C06116=1095.167,-115.821,-48.194,175.111,14.765,152.160
C06117=1095.173,-115.571,-48.203,175.112,14.765,152.159
C06118=1095.179,-115.321,-48.213,175.114,14.765,152.159
C06119=1095.185,-115.071,-48.222,175.116,14.765,152.159
C06120=1095.191,-114.821,-48.232,175.118,14.766,152.158
C06121=1095.198,-114.572,-48.241,175.119,14.766,152.158
C06122=1095.204,-114.322,-48.251,175.121,14.766,152.158
C06123=1095.210,-114.072,-48.261,175.122,14.766,152.157
C06124=1095.216,-113.822,-48.270,175.124,14.767,152.157
C06125=1095.222,-113.572,-48.280,175.126,14.767,152.157
C06126=1095.228,-113.323,-48.289,175.127,14.767,152.156
C06127=1095.234,-113.059,-48.300,175.129,14.767,152.156
C06128=1095.241,-112.794,-48.310,175.130,14.767,152.156
C06129=1095.248,-112.531,-48.320,175.132,14.768,152.156
C06130=1095.254,-112.266,-48.330,175.135,14.768,152.155
C06131=1095.260,-112.016,-48.339,175.136,14.768,152.155
C06132=1095.266,-111.767,-48.349,175.138,14.769,152.155
C06133=1095.273,-111.517,-48.359,175.140,14.769,152.154
C06134=1095.279,-111.268,-48.369,175.141,14.769,152.154
C06135=1095.284,-111.017,-48.379,175.143,14.770,152.154
C06136=1095.290,-110.768,-48.389,175.144,14.770,152.153
C06137=1095.297,-110.518,-48.398,175.146,14.770,152.153
C06138=1095.303,-110.268,-48.408,175.147,14.770,152.153
C06139=1095.309,-110.018,-48.417,175.149,14.771,152.152
C06140=1095.315,-109.768,-48.427,175.151,14.771,152.152
C06141=1095.321,-109.519,-48.436,175.152,14.772,152.152
C06142=1095.328,-109.269,-48.447,175.155,14.772,152.151
C06143=1095.334,-109.020,-48.456,175.156,14.772,152.151
C06144=1095.340,-108.770,-48.466,175.158,14.773,152.151
C06145=1095.346,-108.520,-48.475,175.160,14.773,152.151
C06146=1095.352,-108.270,-48.486,175.161,14.773,152.150
C06147=1095.358,-108.020,-48.495,175.163,14.774,152.150
C06148=1095.364,-107.771,-48.505,175.164,14.773,152.150
C06149=1095.371,-107.521,-48.515,175.166,14.774,152.149
C06150=1095.377,-107.271,-48.525,175.168,14.775,152.149
C06151=1095.383,-107.022,-48.534,175.169,14.774,152.149
C06152=1095.388,-106.771,-48.544,175.171,14.775,152.148
C06153=1095.394,-106.522,-48.554,175.172,14.775,152.148
C06154=1095.401,-106.273,-48.564,175.174,14.776,152.148
C06155=1095.407,-106.023,-48.574,175.177,14.776,152.148
C06156=1095.413,-105.773,-48.583,175.178,14.776,152.147
C06157=1095.419,-105.523,-48.593,175.180,14.777,152.147
C06158=1095.425,-105.274,-48.604,175.181,14.777,152.147
C06159=1095.431,-105.024,-48.613,175.183,14.777,152.146
C06160=1095.438,-104.774,-48.623,175.185,14.778,152.146
C06161=1095.443,-104.524,-48.633,175.186,14.778,152.146
C06162=1095.449,-104.274,-48.643,175.188,14.779,152.146
C06163=1095.456,-104.025,-48.653,175.189,14.778,152.145
C06164=1095.462,-103.775,-48.662,175.191,14.779,152.145
C06165=1095.467,-103.525,-48.673,175.193,14.780,152.145
C06166=1095.474,-103.276,-48.683,175.194,14.780,152.144
C06167=1095.480,-103.026,-48.692,175.196,14.780,152.144
C06168=1095.486,-102.776,-48.702,175.198,14.781,152.144
C06169=1095.491,-102.526,-48.712,175.199,14.781,152.144
C06170=1095.498,-102.277,-48.722,175.201,14.782,152.143
C06171=1095.504,-102.027,-48.732,175.203,14.782,152.143
C06172=1095.510,-101.777,-48.742,175.204,14.782,152.143
C06173=1095.516,-101.528,-48.752,175.206,14.783,152.142
C06174=1095.522,-101.278,-48.762,175.207,14.783,152.142
C06175=1095.528,-101.028,-48.772,175.209,14.783,152.142
C06176=1095.534,-100.779,-48.783,175.211,14.784,152.141
C06177=1095.540,-100.529,-48.792,175.213,14.784,152.141
C06178=1095.546,-100.279,-48.802,175.214,14.784,152.141
C06179=1095.553,-100.030,-48.812,175.216,14.785,152.141
C06180=1095.558,-99.780,-48.822,175.217,14.785,152.140
C06181=1095.565,-99.530,-48.832,175.220,14.785,152.140
C06182=1095.571,-99.281,-48.842,175.222,14.786,152.140
C06183=1095.576,-99.031,-48.852,175.223,14.786,152.140
C06184=1095.583,-98.780,-48.862,175.225,14.787,152.139
C06185=1095.590,-98.531,-48.872,175.227,14.787,152.139
C06186=1095.595,-98.281,-48.882,175.228,14.787,152.139
C06187=1095.602,-98.032,-48.893,175.230,14.788,152.138
C06188=1095.608,-97.782,-48.902,175.231,14.788,152.138
C06189=1095.613,-97.532,-48.912,175.233,14.789,152.138
C06190=1095.620,-97.283,-48.923,175.235,14.790,152.138
C06191=1095.626,-97.009,-48.934,175.237,14.790,152.137
C06192=1095.632,-96.735,-48.945,175.238,14.790,152.137
C06193=1095.639,-96.461,-48.956,175.240,14.791,152.137
C06194=1095.646,-96.187,-48.967,175.242,14.791,152.136
C06195=1095.652,-95.937,-48.978,175.244,14.791,152.136
C06196=1095.658,-95.687,-48.987,175.245,14.792,152.136
C06197=1095.664,-95.438,-48.998,175.247,14.792,152.135
C06198=1095.670,-95.188,-49.008,175.249,14.793,152.135
C06199=1095.675,-94.939,-49.019,175.251,14.794,152.135
C06200=1095.682,-94.689,-49.028,175.252,14.794,152.135
C06201=1095.687,-94.439,-49.039,175.254,14.795,152.134
C06202=1095.694,-94.190,-49.049,175.256,14.795,152.134
C06203=1095.699,-93.940,-49.059,175.257,14.795,152.134
C06204=1095.705,-93.690,-49.069,175.259,14.796,152.133
C06205=1095.711,-93.440,-49.079,175.261,14.796,152.133
C06206=1095.718,-93.190,-49.090,175.262,14.796,152.133
C06207=1095.723,-92.940,-49.100,175.264,14.797,152.133
C06208=1095.730,-92.691,-49.110,175.266,14.798,152.132
C06209=1095.735,-92.441,-49.121,175.267,14.798,152.132
C06210=1095.742,-92.192,-49.131,175.269,14.799,152.132
C06211=1095.747,-91.942,-49.141,175.271,14.799,152.132
C06212=1095.754,-91.693,-49.151,175.272,14.799,152.131
C06213=1095.759,-91.443,-49.162,175.274,14.800,152.131
C06214=1095.766,-91.193,-49.172,175.276,14.800,152.131
C06215=1095.772,-90.943,-49.183,175.278,14.801,152.131
C06216=1095.778,-90.693,-49.193,175.279,14.801,152.130
C06217=1095.784,-90.444,-49.204,175.281,14.802,152.130
C06218=1095.789,-90.194,-49.214,175.283,14.803,152.130
C06219=1095.796,-89.944,-49.224,175.284,14.803,152.130
C06220=1095.802,-89.695,-49.235,175.286,14.804,152.129
C06221=1095.808,-89.445,-49.244,175.287,14.804,152.129
C06222=1095.813,-89.196,-49.255,175.290,14.804,152.129
C06223=1095.820,-88.945,-49.265,175.291,14.805,152.128
C06224=1095.826,-88.696,-49.276,175.293,14.805,152.128
C06225=1095.832,-88.447,-49.286,175.294,14.806,152.128
C06226=1095.838,-88.196,-49.297,175.296,14.806,152.128
C06227=1095.844,-87.947,-49.307,175.297,14.807,152.127
C06228=1095.850,-87.697,-49.317,175.299,14.808,152.127
C06229=1095.856,-87.447,-49.328,175.301,14.808,152.127
C06230=1095.863,-87.198,-49.339,175.302,14.808,152.127
C06231=1095.868,-86.948,-49.349,175.304,14.809,152.126
C06232=1095.874,-86.698,-49.360,175.306,14.809,152.126
C06233=1095.880,-86.449,-49.370,175.308,14.809,152.126
C06234=1095.886,-86.198,-49.380,175.309,14.810,152.125
C06235=1095.893,-85.949,-49.391,175.311,14.811,152.125
C06236=1095.898,-85.699,-49.402,175.313,14.812,152.125
C06237=1095.904,-85.449,-49.412,175.314,14.812,152.125
C06238=1095.910,-85.200,-49.422,175.316,14.812,152.124
C06239=1095.917,-84.950,-49.433,175.318,14.813,152.124
C06240=1095.923,-84.701,-49.443,175.320,14.814,152.124
C06241=1095.929,-84.451,-49.454,175.321,14.814,152.124
C06242=1095.934,-84.201,-49.465,175.323,14.815,152.123
C06243=1095.941,-83.951,-49.475,175.325,14.815,152.123
C06244=1095.947,-83.702,-49.486,175.327,14.816,152.123
C06245=1095.953,-83.452,-49.496,175.328,14.816,152.122
C06246=1095.959,-83.203,-49.506,175.330,14.816,152.122
C06247=1095.965,-82.953,-49.517,175.332,14.817,152.122
C06248=1095.972,-82.703,-49.528,175.334,14.818,152.122
C06249=1095.977,-82.453,-49.538,175.335,14.818,152.121
C06250=1095.983,-82.204,-49.549,175.337,14.819,152.121
C06251=1095.990,-81.954,-49.559,175.339,14.819,152.121
C06252=1095.996,-81.704,-49.571,175.341,14.820,152.121
C06253=1096.001,-81.454,-49.581,175.342,14.820,152.120
C06254=1096.008,-81.205,-49.591,175.344,14.821,152.120
C06255=1096.015,-80.933,-49.603,175.346,14.821,152.120
C06256=1096.021,-80.662,-49.615,175.348,14.822,152.119
C06257=1096.028,-80.390,-49.626,175.350,14.823,152.119
C06258=1096.034,-80.119,-49.638,175.351,14.823,152.119
C06259=1096.041,-79.869,-49.649,175.353,14.823,152.119
C06260=1096.046,-79.619,-49.660,175.354,14.824,152.118
C06261=1096.052,-79.369,-49.670,175.356,14.825,152.118
C06262=1096.058,-79.120,-49.680,175.358,14.826,152.118
C06263=1096.065,-78.870,-49.691,175.360,14.826,152.118
C06264=1096.070,-78.620,-49.702,175.361,14.826,152.117
C06265=1096.076,-78.371,-49.713,175.363,14.827,152.117
C06266=1096.082,-78.121,-49.724,175.365,14.828,152.117
C06267=1096.088,-77.871,-49.735,175.367,14.829,152.117
C06268=1096.094,-77.621,-49.745,175.368,14.829,152.116
C06269=1096.100,-77.372,-49.756,175.370,14.829,152.116
C06270=1096.106,-77.122,-49.767,175.372,14.830,152.116
C06271=1096.112,-76.872,-49.778,175.374,14.831,152.116
C06272=1096.118,-76.623,-49.789,175.375,14.831,152.115
C06273=1096.124,-76.373,-49.800,175.377,14.832,152.115
C06274=1096.130,-76.124,-49.810,175.378,14.832,152.115
C06275=1096.137,-75.874,-49.821,175.380,14.833,152.115
C06276=1096.142,-75.624,-49.832,175.382,14.834,152.114
C06277=1096.148,-75.375,-49.843,175.384,14.834,152.114
C06278=1096.154,-75.125,-49.854,175.385,14.835,152.114
C06279=1096.160,-74.874,-49.864,175.387,14.835,152.113
C06280=1096.166,-74.625,-49.875,175.389,14.836,152.113
C06281=1096.172,-74.376,-49.885,175.391,14.837,152.113
C06282=1096.178,-74.126,-49.897,175.392,14.837,152.113
C06283=1096.184,-73.876,-49.908,175.394,14.838,152.112
C06284=1096.190,-73.627,-49.918,175.396,14.838,152.112
C06285=1096.196,-73.377,-49.929,175.398,14.839,152.112
C06286=1096.202,-73.127,-49.941,175.400,14.840,152.112
C06287=1096.208,-72.877,-49.951,175.401,14.840,152.111
C06288=1096.213,-72.628,-49.962,175.402,14.841,152.111
C06289=1096.218,-72.378,-49.974,175.404,14.842,152.111
C06290=1096.225,-72.128,-49.985,175.406,14.842,152.111
C06291=1096.230,-71.878,-49.996,175.408,14.843,152.111
C06292=1096.236,-71.629,-50.007,175.410,14.844,152.110
C06293=1096.243,-71.379,-50.018,175.411,14.844,152.110
C06294=1096.248,-71.129,-50.029,175.413,14.845,152.110
C06295=1096.254,-70.880,-50.040,175.415,14.845,152.110
C06296=1096.260,-70.630,-50.051,175.417,14.846,152.109
C06297=1096.266,-70.380,-50.062,175.418,14.847,152.109
C06298=1096.272,-70.131,-50.073,175.420,14.848,152.109
C06299=1096.278,-69.881,-50.084,175.421,14.848,152.109
C06300=1096.284,-69.632,-50.096,175.423,14.849,152.108
C06301=1096.290,-69.382,-50.107,175.425,14.850,152.108
C06302=1096.296,-69.133,-50.117,175.427,14.850,152.108
C06303=1096.301,-68.883,-50.128,175.429,14.851,152.108
C06304=1096.308,-68.633,-50.140,175.430,14.852,152.107
C06305=1096.313,-68.383,-50.151,175.432,14.852,152.107
C06306=1096.319,-68.134,-50.162,175.433,14.853,152.107
C06307=1096.325,-67.883,-50.173,175.435,14.853,152.107
C06308=1096.331,-67.634,-50.184,175.437,14.854,152.106
C06309=1096.336,-67.384,-50.195,175.439,14.855,152.106
C06310=1096.343,-67.135,-50.207,175.441,14.856,152.106
C06311=1096.349,-66.885,-50.218,175.443,14.857,152.106
C06312=1096.354,-66.636,-50.229,175.444,14.857,152.106
C06313=1096.361,-66.386,-50.240,175.446,14.858,152.105
C06314=1096.367,-66.136,-50.251,175.447,14.858,152.105
C06315=1096.372,-65.886,-50.263,175.449,14.859,152.105
C06316=1096.378,-65.637,-50.274,175.451,14.860,152.104
C06317=1096.384,-65.387,-50.285,175.453,14.860,152.104
C06318=1096.390,-65.137,-50.296,175.455,14.861,152.104
C06319=1096.396,-64.868,-50.309,175.457,14.862,152.104
C06320=1096.403,-64.598,-50.320,175.459,14.863,152.103
C06321=1096.409,-64.329,-50.333,175.461,14.863,152.103
C06322=1096.416,-64.059,-50.344,175.463,14.864,152.103
C06323=1096.422,-63.811,-50.356,175.464,14.864,152.103
C06324=1096.428,-63.560,-50.367,175.466,14.865,152.102
C06325=1096.433,-63.311,-50.379,175.467,14.866,152.102
C06326=1096.439,-63.061,-50.390,175.469,14.867,152.102
C06327=1096.446,-62.812,-50.401,175.471,14.868,152.102
C06328=1096.451,-62.562,-50.412,175.473,14.868,152.101
C06329=1096.458,-62.312,-50.424,175.475,14.869,152.101
C06330=1096.463,-62.062,-50.434,175.476,14.869,152.101
C06331=1096.469,-61.813,-50.447,175.478,14.870,152.101
C06332=1096.475,-61.563,-50.458,175.479,14.871,152.100
C06333=1096.481,-61.313,-50.469,175.481,14.871,152.100
C06334=1096.487,-61.064,-50.481,175.483,14.872,152.100
C06335=1096.493,-60.814,-50.492,175.485,14.873,152.100
C06336=1096.500,-60.564,-50.503,175.487,14.873,152.099
C06337=1096.505,-60.314,-50.514,175.489,14.875,152.099
C06338=1096.511,-60.065,-50.526,175.490,14.875,152.099
C06339=1096.517,-59.815,-50.537,175.492,14.875,152.099
C06340=1096.523,-59.566,-50.548,175.493,14.876,152.099
C06341=1096.529,-59.316,-50.560,175.495,14.877,152.098
C06342=1096.534,-59.066,-50.571,175.497,14.878,152.098
C06343=1096.541,-58.816,-50.583,175.499,14.878,152.098
C06344=1096.547,-58.567,-50.594,175.501,14.879,152.098
C06345=1096.553,-58.317,-50.606,175.503,14.880,152.097
C06346=1096.559,-58.068,-50.617,175.505,14.881,152.097
C06347=1096.565,-57.818,-50.629,175.506,14.881,152.097
C06348=1096.570,-57.568,-50.640,175.508,14.881,152.096
C06349=1096.577,-57.319,-50.652,175.509,14.883,152.096
C06350=1096.583,-57.069,-50.663,175.511,14.883,152.096
C06351=1096.589,-56.819,-50.675,175.513,14.884,152.096
C06352=1096.594,-56.570,-50.686,175.515,14.885,152.096
C06353=1096.601,-56.320,-50.697,175.517,14.885,152.095
C06354=1096.607,-56.071,-50.709,175.519,14.886,152.095
C06355=1096.612,-55.820,-50.721,175.521,14.887,152.095
C06356=1096.618,-55.572,-50.732,175.522,14.888,152.095
C06357=1096.625,-55.321,-50.744,175.524,14.888,152.094
C06358=1096.631,-55.072,-50.756,175.525,14.888,152.094
C06359=1096.636,-54.822,-50.767,175.527,14.889,152.094
C06360=1096.643,-54.572,-50.779,175.529,14.890,152.094
C06361=1096.649,-54.323,-50.790,175.531,14.891,152.093
C06362=1096.656,-54.073,-50.802,175.533,14.891,152.093
C06363=1096.661,-53.824,-50.813,175.535,14.893,152.093
C06364=1096.667,-53.574,-50.825,175.536,14.893,152.093
C06365=1096.673,-53.324,-50.836,175.538,14.894,152.092
C06366=1096.679,-53.075,-50.849,175.540,14.895,152.092
C06367=1096.685,-52.824,-50.860,175.542,14.895,152.092
C06368=1096.691,-52.576,-50.872,175.543,14.896,152.092
C06369=1096.698,-52.325,-50.883,175.545,14.896,152.091
C06370=1096.703,-52.076,-50.895,175.547,14.897,152.091
C06371=1096.709,-51.826,-50.906,175.549,14.898,152.091
C06372=1096.715,-51.577,-50.918,175.551,14.898,152.091
C06373=1096.721,-51.327,-50.930,175.553,14.899,152.090
C06374=1096.727,-51.077,-50.942,175.555,14.900,152.090
C06375=1096.734,-50.828,-50.953,175.556,14.901,152.090
C06376=1096.739,-50.578,-50.965,175.558,14.901,152.090
C06377=1096.745,-50.329,-50.977,175.560,14.903,152.089
C06378=1096.751,-50.078,-50.988,175.562,14.903,152.089
C06379=1096.757,-49.829,-51.000,175.564,14.904,152.089
C06380=1096.763,-49.579,-51.013,175.565,14.905,152.089
C06381=1096.768,-49.330,-51.024,175.567,14.905,152.088
C06382=1096.774,-49.080,-51.036,175.569,14.906,152.088
C06383=1096.781,-48.812,-51.048,175.571,14.907,152.088
C06384=1096.787,-48.544,-51.061,175.573,14.908,152.088
C06385=1096.794,-48.276,-51.074,175.575,14.909,152.088
C06386=1096.800,-48.008,-51.087,175.576,14.910,152.087
C06387=1096.806,-47.758,-51.099,175.578,14.910,152.087
C06388=1096.811,-47.508,-51.110,175.580,14.911,152.087
C06389=1096.818,-47.259,-51.122,175.582,14.912,152.086
C06390=1096.823,-47.010,-51.134,175.584,14.912,152.086
C06391=1096.829,-46.759,-51.146,175.586,14.913,152.086
C06392=1096.835,-46.510,-51.158,175.587,14.914,152.086
C06393=1096.841,-46.260,-51.170,175.589,14.915,152.086
C06394=1096.847,-46.011,-51.181,175.591,14.916,152.085
C06395=1096.852,-45.761,-51.194,175.593,14.917,152.085
C06396=1096.859,-45.511,-51.206,175.594,14.917,152.085
C06397=1096.864,-45.262,-51.217,175.596,14.917,152.085
C06398=1096.870,-45.012,-51.230,175.598,14.919,152.084
C06399=1096.876,-44.763,-51.241,175.600,14.919,152.084
C06400=1096.882,-44.513,-51.254,175.601,14.920,152.084
C06401=1096.888,-44.263,-51.265,175.603,14.921,152.084
C06402=1096.894,-44.014,-51.277,175.605,14.922,152.083
C06403=1096.900,-43.764,-51.289,175.607,14.922,152.083
C06404=1096.906,-43.514,-51.302,175.609,14.923,152.083
C06405=1096.911,-43.264,-51.313,175.611,14.924,152.083
C06406=1096.918,-43.015,-51.325,175.612,14.925,152.083
C06407=1096.923,-42.766,-51.337,175.614,14.926,152.082
C06408=1096.930,-42.516,-51.349,175.616,14.926,152.082
C06409=1096.936,-42.266,-51.362,175.618,14.927,152.082
C06410=1096.941,-42.016,-51.373,175.620,14.928,152.081
C06411=1096.947,-41.767,-51.385,175.622,14.929,152.081
C06412=1096.953,-41.517,-51.398,175.624,14.929,152.081
C06413=1096.959,-41.268,-51.410,175.626,14.930,152.081
C06414=1096.965,-41.018,-51.422,175.627,14.931,152.081
C06415=1096.971,-40.768,-51.434,175.629,14.932,152.080
C06416=1096.977,-40.519,-51.445,175.631,14.933,152.080
C06417=1096.983,-40.269,-51.458,175.633,14.933,152.080
C06418=1096.989,-40.019,-51.470,175.635,14.934,152.080
C06419=1096.995,-39.770,-51.482,175.637,14.935,152.079
C06420=1097.001,-39.520,-51.495,175.638,14.936,152.079
C06421=1097.007,-39.270,-51.507,175.640,14.936,152.079
C06422=1097.013,-39.021,-51.519,175.642,14.938,152.079
C06423=1097.018,-38.771,-51.531,175.644,14.938,152.078
C06424=1097.024,-38.521,-51.543,175.646,14.939,152.078
C06425=1097.029,-38.272,-51.555,175.648,14.940,152.078
C06426=1097.036,-38.022,-51.567,175.649,14.940,152.078
C06427=1097.042,-37.772,-51.580,175.651,14.941,152.077
C06428=1097.047,-37.523,-51.592,175.653,14.942,152.077
C06429=1097.053,-37.273,-51.605,175.655,14.943,152.077
C06430=1097.059,-37.023,-51.617,175.657,14.944,152.077
C06431=1097.065,-36.775,-51.629,175.659,14.945,152.076
C06432=1097.071,-36.525,-51.641,175.660,14.945,152.076
C06433=1097.077,-36.275,-51.654,175.662,14.946,152.076
C06434=1097.082,-36.026,-51.666,175.664,14.947,152.076
C06435=1097.088,-35.776,-51.679,175.666,14.948,152.076
C06436=1097.094,-35.526,-51.691,175.668,14.949,152.075
C06437=1097.100,-35.276,-51.702,175.669,14.949,152.075
C06438=1097.106,-35.026,-51.715,175.671,14.950,152.075
C06439=1097.112,-34.777,-51.727,175.673,14.951,152.075
C06440=1097.118,-34.527,-51.740,175.675,14.952,152.074
C06441=1097.123,-34.278,-51.752,175.677,14.953,152.074
C06442=1097.129,-34.028,-51.765,175.679,14.954,152.074
C06443=1097.136,-33.779,-51.777,175.680,14.954,152.074
C06444=1097.142,-33.529,-51.790,175.682,14.955,152.073
C06445=1097.147,-33.280,-51.802,175.684,14.956,152.073
C06446=1097.153,-33.030,-51.814,175.686,14.956,152.073
C06447=1097.159,-32.762,-51.827,175.688,14.957,152.073
C06448=1097.165,-32.494,-51.841,175.691,14.958,152.072
C06449=1097.172,-32.226,-51.854,175.692,14.960,152.072
C06450=1097.178,-31.959,-51.868,175.694,14.960,152.072
C06451=1097.184,-31.709,-51.880,175.696,14.961,152.072
C06452=1097.189,-31.460,-51.892,175.698,14.962,152.071
C06453=1097.195,-31.210,-51.905,175.700,14.963,152.071
C06454=1097.201,-30.960,-51.918,175.702,14.963,152.071
C06455=1097.207,-30.710,-51.930,175.703,14.964,152.071
C06456=1097.213,-30.461,-51.942,175.705,14.965,152.070
C06457=1097.219,-30.211,-51.954,175.707,14.966,152.070
C06458=1097.225,-29.961,-51.967,175.709,14.967,152.070
C06459=1097.231,-29.712,-51.980,175.711,14.967,152.070
C06460=1097.237,-29.462,-51.993,175.713,14.968,152.070
C06461=1097.242,-29.213,-52.005,175.714,14.969,152.069
C06462=1097.248,-28.963,-52.017,175.716,14.970,152.069
C06463=1097.254,-28.713,-52.030,175.718,14.970,152.069
C06464=1097.260,-28.464,-52.042,175.720,14.971,152.069
C06465=1097.266,-28.214,-52.056,175.723,14.972,152.068
C06466=1097.272,-27.965,-52.068,175.725,14.973,152.068
C06467=1097.278,-27.715,-52.080,175.726,14.974,152.068
C06468=1097.284,-27.465,-52.093,175.728,14.975,152.068
C06469=1097.289,-27.215,-52.106,175.730,14.976,152.067
C06470=1097.296,-26.966,-52.118,175.732,14.977,152.067
C06471=1097.302,-26.716,-52.131,175.734,14.977,152.067
C06472=1097.307,-26.467,-52.144,175.736,14.978,152.067
C06473=1097.313,-26.217,-52.156,175.738,14.979,152.066
C06474=1097.319,-25.968,-52.169,175.739,14.980,152.066
C06475=1097.325,-25.718,-52.182,175.741,14.981,152.066
C06476=1097.331,-25.468,-52.195,175.743,14.981,152.066
C06477=1097.336,-25.219,-52.207,175.745,14.982,152.065
C06478=1097.342,-24.970,-52.220,175.747,14.983,152.065
C06479=1097.348,-24.720,-52.233,175.748,14.984,152.065
C06480=1097.354,-24.470,-52.245,175.750,14.984,152.065
C06481=1097.360,-24.220,-52.258,175.752,14.986,152.065
C06482=1097.365,-23.971,-52.271,175.755,14.987,152.064
C06483=1097.371,-23.721,-52.284,175.756,14.988,152.064
C06484=1097.377,-23.471,-52.296,175.758,14.988,152.064
C06485=1097.383,-23.222,-52.310,175.760,14.989,152.063
C06486=1097.389,-22.972,-52.322,175.762,14.990,152.063
C06487=1097.395,-22.722,-52.335,175.764,14.991,152.063
C06488=1097.400,-22.474,-52.348,175.766,14.991,152.063
C06489=1097.406,-22.224,-52.360,175.767,14.993,152.063
C06490=1097.411,-21.974,-52.373,175.769,14.993,152.062
C06491=1097.418,-21.725,-52.387,175.771,14.994,152.062
C06492=1097.424,-21.475,-52.399,175.773,14.995,152.062
C06493=1097.430,-21.225,-52.412,175.775,14.995,152.062
C06494=1097.436,-20.975,-52.425,175.777,14.996,152.061
C06495=1097.441,-20.726,-52.437,175.780,14.997,152.061
C06496=1097.447,-20.477,-52.451,175.781,14.998,152.061
C06497=1097.452,-20.227,-52.464,175.783,14.999,152.060
C06498=1097.459,-19.978,-52.477,175.785,15.000,152.060
C06499=1097.465,-19.728,-52.489,175.787,15.001,152.060
C06500=1097.470,-19.478,-52.502,175.789,15.002,152.060
C06501=1097.477,-19.229,-52.515,175.790,15.002,152.060
C06502=1097.482,-18.978,-52.528,175.792,15.003,152.059
C06503=1097.488,-18.729,-52.542,175.794,15.004,152.059
C06504=1097.494,-18.479,-52.554,175.796,15.005,152.059
C06505=1097.500,-18.231,-52.567,175.798,15.005,152.059
C06506=1097.505,-17.981,-52.580,175.801,15.007,152.058
C06507=1097.511,-17.731,-52.593,175.803,15.007,152.058
C06508=1097.517,-17.481,-52.606,175.804,15.008,152.058
C06509=1097.523,-17.232,-52.619,175.806,15.009,152.058
C06510=1097.529,-16.982,-52.632,175.808,15.010,152.057
C06511=1097.535,-16.714,-52.647,175.810,15.011,152.057
C06512=1097.542,-16.445,-52.660,175.812,15.012,152.057
C06513=1097.548,-16.177,-52.675,175.814,15.013,152.057
C06514=1097.554,-15.908,-52.688,175.816,15.014,152.056
C06515=1097.560,-15.659,-52.701,175.818,15.014,152.056
C06516=1097.566,-15.409,-52.714,175.820,15.015,152.056
C06517=1097.572,-15.159,-52.728,175.822,15.016,152.056
C06518=1097.578,-14.910,-52.740,175.824,15.017,152.055
C06519=1097.584,-14.660,-52.754,175.826,15.017,152.055
C06520=1097.589,-14.410,-52.767,175.828,15.019,152.055
C06521=1097.595,-14.161,-52.780,175.830,15.019,152.054
C06522=1097.601,-13.911,-52.794,175.832,15.020,152.054
C06523=1097.607,-13.661,-52.806,175.834,15.021,152.054
C06524=1097.613,-13.412,-52.820,175.836,15.022,152.054
C06525=1097.618,-13.162,-52.833,175.838,15.022,152.053
C06526=1097.624,-12.913,-52.846,175.839,15.023,152.053
C06527=1097.630,-12.663,-52.860,175.841,15.024,152.053
C06528=1097.636,-12.413,-52.872,175.844,15.026,152.053
C06529=1097.642,-12.164,-52.886,175.846,15.026,152.053
C06530=1097.647,-11.914,-52.900,175.847,15.027,152.052
C06531=1097.653,-11.664,-52.912,175.849,15.028,152.052
C06532=1097.659,-11.415,-52.926,175.851,15.028,152.052
C06533=1097.665,-11.166,-52.939,175.853,15.029,152.052
C06534=1097.671,-10.916,-52.952,175.855,15.030,152.051
C06535=1097.676,-10.667,-52.965,175.857,15.031,152.051
C06536=1097.682,-10.418,-52.979,175.860,15.032,152.051
C06537=1097.687,-10.167,-52.992,175.861,15.033,152.050
C06538=1097.693,-9.918,-53.005,175.863,15.033,152.050
C06539=1097.699,-9.669,-53.019,175.865,15.034,152.050
C06540=1097.705,-9.418,-53.032,175.867,15.035,152.050
C06541=1097.711,-9.169,-53.045,175.869,15.036,152.050
C06542=1097.717,-8.919,-53.059,175.871,15.037,152.049
C06543=1097.723,-8.670,-53.072,175.872,15.038,152.049
C06544=1097.728,-8.420,-53.085,175.875,15.039,152.049
C06545=1097.734,-8.170,-53.099,175.877,15.040,152.049
C06546=1097.740,-7.921,-53.112,175.879,15.040,152.048
C06547=1097.746,-7.672,-53.126,175.881,15.041,152.048
C06548=1097.751,-7.421,-53.139,175.883,15.042,152.048
C06549=1097.758,-7.172,-53.152,175.884,15.043,152.048
C06550=1097.763,-6.923,-53.166,175.886,15.043,152.047
C06551=1097.769,-6.673,-53.179,175.889,15.045,152.047
C06552=1097.775,-6.424,-53.193,175.891,15.045,152.047
C06553=1097.781,-6.174,-53.206,175.893,15.046,152.046
C06554=1097.786,-5.924,-53.220,175.895,15.047,152.046
C06555=1097.792,-5.675,-53.233,175.897,15.048,152.046
C06556=1097.798,-5.425,-53.247,175.898,15.048,152.046
C06557=1097.804,-5.176,-53.260,175.900,15.049,152.045
C06558=1097.809,-4.927,-53.274,175.903,15.050,152.045
C06559=1097.816,-4.677,-53.287,175.905,15.051,152.045
C06560=1097.822,-4.427,-53.301,175.907,15.052,152.045
C06561=1097.828,-4.177,-53.314,175.909,15.053,152.044
C06562=1097.833,-3.928,-53.328,175.910,15.053,152.044
C06563=1097.839,-3.678,-53.341,175.912,15.054,152.044
C06564=1097.845,-3.429,-53.355,175.914,15.055,152.044
C06565=1097.851,-3.180,-53.368,175.917,15.056,152.043
C06566=1097.857,-2.930,-53.382,175.919,15.057,152.043
C06567=1097.862,-2.680,-53.396,175.921,15.058,152.043
C06568=1097.868,-2.431,-53.409,175.923,15.058,152.043
C06569=1097.874,-2.182,-53.423,175.924,15.059,152.042
C06570=1097.879,-1.932,-53.437,175.926,15.060,152.042
C06571=1097.885,-1.682,-53.451,175.929,15.061,152.042
C06572=1097.891,-1.432,-53.464,175.931,15.062,152.041
C06573=1097.897,-1.182,-53.478,175.933,15.063,152.041
C06574=1097.902,-0.933,-53.491,175.935,15.063,152.041
C06575=1097.908,-0.663,-53.506,175.937,15.065,152.041
C06576=1097.915,-0.392,-53.521,175.939,15.066,152.040
C06577=1097.921,-0.123,-53.535,175.941,15.066,152.040
C06578=1097.927,0.148,-53.551,175.944,15.068,152.040
C06579=1097.933,0.398,-53.565,175.946,15.068,152.040
C06580=1097.938,0.647,-53.578,175.947,15.069,152.039
C06581=1097.944,0.897,-53.592,175.949,15.070,152.039
C06582=1097.950,1.145,-53.606,175.951,15.071,152.039
C06583=1097.956,1.395,-53.620,175.953,15.071,152.039
C06584=1097.961,1.645,-53.634,175.956,15.073,152.038
C06585=1097.967,1.894,-53.647,175.958,15.073,152.038
C06586=1097.973,2.143,-53.661,175.959,15.074,152.038
C06587=1097.979,2.394,-53.675,175.961,15.075,152.037
C06588=1097.984,2.643,-53.689,175.963,15.076,152.037
C06589=1097.991,2.893,-53.703,175.966,15.077,152.037
C06590=1097.996,3.142,-53.716,175.968,15.078,152.037
C06591=1098.001,3.392,-53.730,175.970,15.078,152.036
C06592=1098.007,3.641,-53.744,175.971,15.079,152.036
C06593=1098.013,3.892,-53.758,175.974,15.079,152.036
C06594=1098.020,4.140,-53.772,175.976,15.081,152.035
C06595=1098.025,4.390,-53.786,175.978,15.081,152.035
C06596=1098.030,4.639,-53.800,175.980,15.082,152.035
C06597=1098.036,4.889,-53.814,175.982,15.083,152.035
C06598=1098.041,5.139,-53.828,175.984,15.084,152.034
C06599=1098.048,5.389,-53.841,175.986,15.084,152.034
C06600=1098.054,5.638,-53.855,175.988,15.086,152.034
C06601=1098.060,5.887,-53.870,175.990,15.087,152.034
C06602=1098.065,6.137,-53.884,175.992,15.087,152.033
C06603=1098.070,6.386,-53.898,175.994,15.088,152.033
C06604=1098.077,6.636,-53.912,175.996,15.089,152.033
C06605=1098.083,6.886,-53.925,175.999,15.090,152.033
C06606=1098.089,7.135,-53.940,176.001,15.090,152.032
C06607=1098.094,7.384,-53.954,176.003,15.091,152.032
C06608=1098.100,7.635,-53.968,176.005,15.092,152.032
C06609=1098.106,7.884,-53.982,176.006,15.093,152.031
C06610=1098.111,8.133,-53.996,176.009,15.094,152.031
C06611=1098.117,8.383,-54.010,176.011,15.095,152.031
C06612=1098.124,8.633,-54.024,176.013,15.095,152.031
C06613=1098.129,8.882,-54.038,176.015,15.096,152.030
C06614=1098.135,9.131,-54.052,176.017,15.096,152.030
C06615=1098.140,9.381,-54.066,176.020,15.098,152.030
C06616=1098.146,9.631,-54.080,176.021,15.098,152.029
C06617=1098.152,9.880,-54.095,176.023,15.099,152.029
C06618=1098.158,10.130,-54.109,176.025,15.100,152.029
C06619=1098.163,10.379,-54.123,176.027,15.101,152.029
C06620=1098.170,10.629,-54.138,176.030,15.102,152.028
C06621=1098.176,10.878,-54.151,176.032,15.102,152.028
C06622=1098.181,11.128,-54.165,176.034,15.103,152.028
C06623=1098.188,11.377,-54.180,176.036,15.104,152.027
C06624=1098.193,11.627,-54.193,176.038,15.105,152.027
C06625=1098.199,11.876,-54.207,176.040,15.106,152.027
C06626=1098.204,12.125,-54.222,176.042,15.106,152.026
C06627=1098.210,12.376,-54.236,176.044,15.107,152.026
C06628=1098.216,12.625,-54.251,176.046,15.108,152.026
C06629=1098.222,12.874,-54.265,176.049,15.109,152.026
C06630=1098.228,13.124,-54.280,176.051,15.110,152.025
C06631=1098.234,13.373,-54.293,176.053,15.110,152.025
C06632=1098.239,13.623,-54.307,176.055,15.111,152.025
C06633=1098.245,13.873,-54.322,176.057,15.111,152.024
C06634=1098.252,14.122,-54.335,176.059,15.113,152.024
C06635=1098.258,14.372,-54.350,176.061,15.114,152.024
C06636=1098.263,14.621,-54.365,176.063,15.114,152.023
C06637=1098.269,14.870,-54.379,176.065,15.115,152.023
C06638=1098.274,15.120,-54.393,176.068,15.116,152.023
C06639=1098.281,15.393,-54.409,176.070,15.117,152.023
C06640=1098.287,15.664,-54.425,176.072,15.117,152.022
C06641=1098.293,15.937,-54.441,176.075,15.118,152.022
C06642=1098.300,16.208,-54.456,176.077,15.119,152.022
C06643=1098.306,16.459,-54.470,176.079,15.120,152.021
C06644=1098.312,16.707,-54.485,176.081,15.121,152.021
C06645=1098.316,16.957,-54.499,176.083,15.121,152.021
C06646=1098.323,17.207,-54.514,176.085,15.122,152.021
C06647=1098.328,17.457,-54.528,176.088,15.123,152.020
C06648=1098.334,17.706,-54.543,176.090,15.124,152.020
C06649=1098.340,17.956,-54.557,176.092,15.124,152.020
C06650=1098.346,18.205,-54.572,176.094,15.125,152.019
C06651=1098.351,18.454,-54.586,176.096,15.126,152.019
C06652=1098.357,18.704,-54.601,176.098,15.127,152.019
C06653=1098.363,18.953,-54.616,176.100,15.128,152.018
C06654=1098.369,19.204,-54.630,176.102,15.128,152.018
C06655=1098.375,19.452,-54.644,176.104,15.129,152.018
C06656=1098.380,19.702,-54.658,176.107,15.130,152.018
C06657=1098.386,19.952,-54.673,176.109,15.131,152.017
C06658=1098.392,20.201,-54.688,176.111,15.131,152.017
C06659=1098.397,20.451,-54.702,176.113,15.132,152.017
C06660=1098.403,20.700,-54.717,176.115,15.133,152.016
C06661=1098.409,20.949,-54.732,176.118,15.134,152.016
C06662=1098.415,21.199,-54.746,176.120,15.134,152.016
C06663=1098.420,21.449,-54.761,176.121,15.135,152.015
C06664=1098.426,21.698,-54.776,176.124,15.137,152.015
C06665=1098.432,21.948,-54.790,176.126,15.137,152.015
C06666=1098.438,22.197,-54.805,176.128,15.138,152.014
C06667=1098.444,22.447,-54.820,176.130,15.138,152.014
C06668=1098.449,22.696,-54.834,176.133,15.140,152.014
C06669=1098.455,22.945,-54.849,176.135,15.140,152.013
C06670=1098.460,23.195,-54.864,176.137,15.141,152.013
C06671=1098.466,23.444,-54.879,176.139,15.141,152.013
C06672=1098.472,23.695,-54.893,176.142,15.142,152.013
C06673=1098.478,23.944,-54.908,176.143,15.143,152.012
C06674=1098.484,24.194,-54.923,176.145,15.144,152.012
C06675=1098.489,24.442,-54.938,176.148,15.145,152.012
C06676=1098.495,24.692,-54.952,176.150,15.145,152.011
C06677=1098.501,24.942,-54.967,176.152,15.146,152.011
C06678=1098.506,25.191,-54.982,176.154,15.146,152.011
C06679=1098.513,25.441,-54.997,176.157,15.148,152.010
C06680=1098.518,25.690,-55.012,176.159,15.149,152.010
C06681=1098.524,25.940,-55.026,176.161,15.149,152.010
C06682=1098.530,26.189,-55.041,176.163,15.150,152.009
C06683=1098.536,26.439,-55.056,176.166,15.151,152.009
C06684=1098.541,26.688,-55.071,176.168,15.151,152.009
C06685=1098.547,26.938,-55.086,176.170,15.152,152.008
C06686=1098.553,27.187,-55.101,176.171,15.153,152.008
C06687=1098.559,27.437,-55.116,176.174,15.154,152.008
C06688=1098.564,27.686,-55.130,176.176,15.154,152.008
C06689=1098.570,27.936,-55.145,176.179,15.155,152.007
C06690=1098.576,28.185,-55.160,176.181,15.156,152.007
C06691=1098.582,28.435,-55.175,176.183,15.157,152.007
C06692=1098.587,28.684,-55.190,176.185,15.157,152.006
C06693=1098.594,28.934,-55.205,176.187,15.158,152.006
C06694=1098.599,29.183,-55.220,176.190,15.159,152.006
C06695=1098.604,29.432,-55.235,176.192,15.159,152.005
C06696=1098.610,29.682,-55.250,176.194,15.160,152.005
C06697=1098.616,29.931,-55.265,176.197,15.161,152.004
C06698=1098.622,30.181,-55.280,176.199,15.162,152.004
C06699=1098.627,30.430,-55.295,176.201,15.162,152.004
C06700=1098.633,30.680,-55.310,176.203,15.163,152.004
C06701=1098.639,30.929,-55.325,176.205,15.164,152.003
C06702=1098.644,31.179,-55.340,176.208,15.164,152.003
C06703=1098.651,31.452,-55.357,176.210,15.166,152.003
C06704=1098.657,31.726,-55.373,176.212,15.166,152.002
C06705=1098.664,32.000,-55.390,176.215,15.167,152.002
C06706=1098.669,32.273,-55.406,176.217,15.168,152.001
C06707=1098.675,32.523,-55.422,176.219,15.168,152.001
C06708=1098.681,32.772,-55.436,176.222,15.169,152.001
C06709=1098.687,33.022,-55.452,176.224,15.170,152.001
C06710=1098.692,33.271,-55.466,176.226,15.170,152.000
C06711=1098.698,33.521,-55.482,176.229,15.172,152.000
C06712=1098.704,33.770,-55.496,176.231,15.172,152.000
C06713=1098.709,34.020,-55.512,176.233,15.173,151.999
C06714=1098.716,34.269,-55.527,176.235,15.173,151.999
C06715=1098.721,34.519,-55.542,176.238,15.174,151.998
C06716=1098.728,34.768,-55.558,176.240,15.175,151.998
C06717=1098.733,35.017,-55.573,176.242,15.175,151.998
C06718=1098.738,35.267,-55.588,176.245,15.177,151.997
C06719=1098.745,35.517,-55.603,176.247,15.177,151.997
C06720=1098.750,35.766,-55.619,176.249,15.178,151.997
C06721=1098.756,36.016,-55.634,176.252,15.178,151.996
C06722=1098.761,36.265,-55.649,176.253,15.179,151.996
C06723=1098.768,36.514,-55.664,176.256,15.179,151.996
C06724=1098.773,36.764,-55.680,176.257,15.180,151.995
C06725=1098.778,37.013,-55.695,176.260,15.181,151.995
C06726=1098.785,37.263,-55.710,176.263,15.181,151.995
C06727=1098.790,37.512,-55.725,176.265,15.182,151.994
C06728=1098.796,37.762,-55.740,176.267,15.183,151.994
C06729=1098.802,38.011,-55.756,176.269,15.184,151.994
C06730=1098.807,38.260,-55.772,176.272,15.184,151.993
C06731=1098.813,38.510,-55.787,176.274,15.185,151.993
C06732=1098.819,38.760,-55.802,176.276,15.186,151.993
C06733=1098.825,39.009,-55.818,176.278,15.186,151.992
C06734=1098.830,39.259,-55.834,176.281,15.187,151.992
C06735=1098.836,39.507,-55.848,176.283,15.188,151.992
C06736=1098.842,39.757,-55.864,176.285,15.188,151.991
C06737=1098.848,40.007,-55.880,176.288,15.190,151.991
C06738=1098.853,40.256,-55.895,176.290,15.190,151.990
C06739=1098.859,40.506,-55.910,176.292,15.190,151.990
C06740=1098.864,40.754,-55.926,176.295,15.192,151.990
C06741=1098.870,41.004,-55.941,176.297,15.192,151.989
C06742=1098.876,41.254,-55.957,176.299,15.193,151.989
C06743=1098.881,41.504,-55.972,176.301,15.193,151.989
C06744=1098.887,41.753,-55.988,176.304,15.194,151.988
C06745=1098.893,42.003,-56.003,176.306,15.195,151.988
C06746=1098.898,42.252,-56.019,176.308,15.195,151.988
C06747=1098.904,42.501,-56.035,176.311,15.196,151.987
C06748=1098.910,42.751,-56.050,176.313,15.196,151.987
C06749=1098.916,42.999,-56.066,176.315,15.197,151.986
C06750=1098.921,43.249,-56.081,176.318,15.198,151.986
C06751=1098.927,43.499,-56.097,176.320,15.198,151.986
C06752=1098.933,43.749,-56.113,176.322,15.199,151.986
C06753=1098.938,43.998,-56.128,176.325,15.200,151.985
C06754=1098.944,44.247,-56.144,176.327,15.200,151.985
C06755=1098.950,44.496,-56.159,176.329,15.201,151.984
C06756=1098.955,44.746,-56.175,176.332,15.202,151.984
C06757=1098.961,44.996,-56.191,176.334,15.203,151.984
C06758=1098.966,45.245,-56.206,176.337,15.204,151.983
C06759=1098.972,45.494,-56.222,176.339,15.204,151.983
C06760=1098.978,45.744,-56.238,176.341,15.205,151.983
C06761=1098.983,45.993,-56.254,176.344,15.205,151.982
C06762=1098.989,46.243,-56.269,176.346,15.206,151.982
C06763=1098.995,46.492,-56.285,176.348,15.207,151.982
C06764=1099.000,46.741,-56.301,176.351,15.207,151.981
C06765=1099.006,46.991,-56.317,176.353,15.208,151.981
C06766=1099.012,47.241,-56.332,176.355,15.208,151.980
C06767=1099.018,47.514,-56.350,176.358,15.209,151.980
C06768=1099.024,47.788,-56.367,176.360,15.210,151.980
C06769=1099.030,48.061,-56.385,176.363,15.210,151.979
C06770=1099.036,48.335,-56.402,176.366,15.212,151.979
C06771=1099.042,48.585,-56.418,176.368,15.212,151.978
C06772=1099.048,48.834,-56.434,176.370,15.212,151.978
C06773=1099.053,49.083,-56.449,176.373,15.213,151.978
C06774=1099.059,49.333,-56.466,176.375,15.214,151.977
C06775=1099.064,49.583,-56.481,176.377,15.214,151.977
C06776=1099.070,49.832,-56.497,176.380,15.215,151.976
C06777=1099.076,50.081,-56.513,176.382,15.216,151.976
C06778=1099.081,50.331,-56.529,176.384,15.216,151.976
C06779=1099.087,50.580,-56.545,176.387,15.217,151.975
C06780=1099.093,50.829,-56.561,176.389,15.217,151.975
C06781=1099.098,51.079,-56.576,176.392,15.219,151.975
C06782=1099.104,51.328,-56.593,176.394,15.219,151.974
C06783=1099.110,51.577,-56.609,176.396,15.219,151.974
C06784=1099.116,51.827,-56.625,176.399,15.220,151.973
C06785=1099.122,52.077,-56.641,176.402,15.221,151.973
C06786=1099.127,52.325,-56.657,176.403,15.221,151.973
C06787=1099.133,52.575,-56.672,176.406,15.222,151.972
C06788=1099.139,52.825,-56.688,176.409,15.222,151.972
C06789=1099.144,53.074,-56.705,176.411,15.223,151.971
C06790=1099.150,53.324,-56.721,176.414,15.224,151.971
C06791=1099.155,53.573,-56.737,176.416,15.224,151.971
C06792=1099.161,53.822,-56.753,176.418,15.225,151.970
C06793=1099.167,54.072,-56.769,176.421,15.226,151.970
C06794=1099.172,54.322,-56.785,176.423,15.226,151.969
C06795=1099.178,54.571,-56.801,176.426,15.227,151.969
C06796=1099.184,54.820,-56.817,176.428,15.227,151.969
C06797=1099.190,55.070,-56.834,176.430,15.227,151.968
C06798=1099.196,55.318,-56.849,176.433,15.229,151.968
C06799=1099.201,55.569,-56.866,176.435,15.229,151.968
C06800=1099.206,55.818,-56.882,176.437,15.229,151.967
C06801=1099.212,56.067,-56.898,176.440,15.230,151.967
C06802=1099.218,56.317,-56.914,176.442,15.230,151.966
C06803=1099.224,56.566,-56.931,176.445,15.231,151.966
C06804=1099.230,56.815,-56.947,176.448,15.232,151.965
C06805=1099.236,57.065,-56.962,176.450,15.232,151.965
C06806=1099.241,57.315,-56.979,176.453,15.233,151.965
C06807=1099.246,57.564,-56.995,176.455,15.233,151.964
C06808=1099.252,57.813,-57.011,176.457,15.233,151.964
C06809=1099.258,58.062,-57.028,176.460,15.234,151.963
C06810=1099.264,58.312,-57.044,176.462,15.235,151.963
C06811=1099.270,58.561,-57.060,176.465,15.235,151.962
C06812=1099.276,58.811,-57.077,176.467,15.236,151.962
C06813=1099.281,59.060,-57.093,176.469,15.237,151.962
C06814=1099.287,59.309,-57.110,176.472,15.237,151.961
C06815=1099.293,59.559,-57.126,176.475,15.238,151.961
C06816=1099.299,59.808,-57.142,176.477,15.238,151.960
C06817=1099.305,60.058,-57.158,176.480,15.239,151.960
C06818=1099.310,60.308,-57.174,176.482,15.239,151.959
C06819=1099.316,60.557,-57.191,176.485,15.240,151.959
C06820=1099.322,60.806,-57.207,176.487,15.240,151.959
C06821=1099.328,61.056,-57.223,176.490,15.240,151.958
C06822=1099.333,61.305,-57.240,176.492,15.241,151.958
C06823=1099.339,61.555,-57.256,176.495,15.241,151.957
C06824=1099.345,61.803,-57.273,176.497,15.242,151.957
C06825=1099.351,62.053,-57.290,176.500,15.243,151.957
C06826=1099.357,62.302,-57.306,176.502,15.243,151.956
C06827=1099.363,62.552,-57.323,176.505,15.244,151.956
C06828=1099.369,62.801,-57.339,176.507,15.244,151.955
C06829=1099.374,63.051,-57.355,176.509,15.244,151.955
C06830=1099.380,63.300,-57.371,176.512,15.245,151.954
C06831=1099.386,63.574,-57.390,176.515,15.245,151.954
C06832=1099.393,63.847,-57.408,176.518,15.246,151.953
C06833=1099.400,64.120,-57.426,176.521,15.247,151.953
C06834=1099.405,64.394,-57.444,176.523,15.247,151.952
C06835=1099.411,64.643,-57.460,176.526,15.248,151.952
C06836=1099.417,64.892,-57.478,176.528,15.248,151.952
C06837=1099.423,65.142,-57.494,176.531,15.248,151.951
C06838=1099.429,65.391,-57.510,176.534,15.249,151.951
C06839=1099.434,65.641,-57.527,176.536,15.249,151.950
C06840=1099.440,65.890,-57.543,176.539,15.250,151.950
C06841=1099.445,66.140,-57.560,176.541,15.251,151.949
C06842=1099.451,66.388,-57.577,176.543,15.250,151.949
C06843=1099.457,66.638,-57.594,176.546,15.251,151.948
C06844=1099.462,66.887,-57.610,176.549,15.252,151.948
C06845=1099.468,67.137,-57.626,176.551,15.252,151.948
C06846=1099.474,67.386,-57.643,176.554,15.253,151.947
C06847=1099.480,67.635,-57.660,176.556,15.253,151.947
C06848=1099.485,67.885,-57.677,176.559,15.254,151.946
C06849=1099.491,68.134,-57.693,176.561,15.254,151.946
C06850=1099.496,68.384,-57.710,176.564,15.255,151.945
C06851=1099.503,68.632,-57.727,176.566,15.255,151.945
C06852=1099.508,68.882,-57.744,176.569,15.255,151.944
C06853=1099.514,69.131,-57.760,176.572,15.256,151.944
C06854=1099.519,69.381,-57.777,176.574,15.256,151.943
C06855=1099.525,69.630,-57.794,176.577,15.257,151.943
C06856=1099.530,69.879,-57.811,176.579,15.257,151.943
C06857=1099.537,70.130,-57.828,176.581,15.257,151.942
C06858=1099.542,70.379,-57.845,176.584,15.258,151.942
C06859=1099.548,70.628,-57.862,176.587,15.258,151.941
C06860=1099.554,70.878,-57.878,176.590,15.259,151.941
C06861=1099.559,71.127,-57.896,176.592,15.259,151.940
C06862=1099.565,71.376,-57.912,176.595,15.260,151.940
C06863=1099.570,71.626,-57.929,176.597,15.261,151.939
C06864=1099.576,71.875,-57.946,176.600,15.260,151.939
C06865=1099.582,72.124,-57.963,176.603,15.261,151.938
C06866=1099.587,72.373,-57.980,176.605,15.262,151.938
C06867=1099.593,72.622,-57.997,176.608,15.263,151.938
C06868=1099.598,72.872,-58.013,176.610,15.262,151.937
C06869=1099.605,73.122,-58.031,176.613,15.263,151.937
C06870=1099.611,73.371,-58.048,176.615,15.264,151.936
C06871=1099.616,73.620,-58.065,176.618,15.264,151.936
C06872=1099.621,73.870,-58.082,176.621,15.264,151.935
C06873=1099.627,74.119,-58.099,176.623,15.265,151.935
C06874=1099.633,74.368,-58.116,176.626,15.265,151.934
C06875=1099.638,74.617,-58.133,176.629,15.265,151.934
C06876=1099.644,74.867,-58.150,176.631,15.266,151.933
C06877=1099.650,75.116,-58.168,176.634,15.267,151.933
C06878=1099.656,75.366,-58.184,176.636,15.266,151.932
C06879=1099.662,75.615,-58.201,176.639,15.267,151.932
C06880=1099.667,75.864,-58.218,176.641,15.268,151.931
C06881=1099.672,76.113,-58.236,176.645,15.268,151.931
C06882=1099.678,76.363,-58.252,176.647,15.268,151.930
C06883=1099.684,76.612,-58.270,176.649,15.269,151.930
C06884=1099.690,76.862,-58.287,176.652,15.269,151.929
C06885=1099.696,77.111,-58.304,176.654,15.269,151.929
C06886=1099.701,77.361,-58.321,176.658,15.270,151.928
C06887=1099.707,77.610,-58.338,176.660,15.270,151.928
C06888=1099.712,77.859,-58.356,176.662,15.270,151.928
C06889=1099.719,78.109,-58.372,176.665,15.271,151.927
C06890=1099.724,78.358,-58.390,176.668,15.271,151.927
C06891=1099.730,78.607,-58.407,176.671,15.272,151.926
C06892=1099.735,78.856,-58.424,176.673,15.272,151.926
C06893=1099.741,79.105,-58.442,176.676,15.272,151.925
C06894=1099.747,79.356,-58.459,176.679,15.273,151.925
C06895=1099.753,79.629,-58.478,176.682,15.273,151.924
C06896=1099.759,79.902,-58.497,176.684,15.273,151.924
C06897=1099.765,80.175,-58.516,176.687,15.274,151.923
C06898=1099.771,80.448,-58.535,176.691,15.274,151.922
C06899=1099.777,80.697,-58.552,176.693,15.275,151.922
C06900=1099.783,80.947,-58.570,176.696,15.275,151.922
C06901=1099.788,81.197,-58.587,176.698,15.275,151.921
C06902=1099.794,81.446,-58.604,176.701,15.276,151.921
C06903=1099.799,81.695,-58.622,176.704,15.276,151.920
C06904=1099.806,81.944,-58.640,176.706,15.276,151.920
C06905=1099.811,82.194,-58.657,176.709,15.277,151.919
C06906=1099.816,82.443,-58.674,176.711,15.277,151.919
C06907=1099.822,82.692,-58.692,176.715,15.278,151.918
C06908=1099.827,82.941,-58.709,176.717,15.278,151.918
C06909=1099.833,83.192,-58.726,176.720,15.278,151.917
C06910=1099.839,83.441,-58.744,176.722,15.279,151.917
C06911=1099.845,83.689,-58.761,176.725,15.279,151.916
C06912=1099.851,83.939,-58.779,176.728,15.279,151.916
C06913=1099.856,84.188,-58.796,176.730,15.279,151.915
C06914=1099.862,84.437,-58.814,176.733,15.280,151.915
C06915=1099.867,84.687,-58.831,176.736,15.280,151.914
C06916=1099.873,84.937,-58.849,176.739,15.280,151.913
C06917=1099.879,85.186,-58.866,176.741,15.281,151.913
C06918=1099.884,85.435,-58.884,176.744,15.281,151.912
C06919=1099.891,85.684,-58.902,176.747,15.281,151.912
C06920=1099.896,85.933,-58.919,176.750,15.282,151.911
C06921=1099.902,86.182,-58.937,176.752,15.282,151.911
C06922=1099.907,86.431,-58.955,176.755,15.283,151.910
C06923=1099.913,86.682,-58.972,176.758,15.283,151.910
C06924=1099.918,86.931,-58.989,176.760,15.283,151.909
C06925=1099.924,87.180,-59.007,176.763,15.283,151.909
C06926=1099.930,87.430,-59.025,176.766,15.283,151.908
C06927=1099.936,87.679,-59.042,176.769,15.284,151.908
C06928=1099.941,87.928,-59.060,176.771,15.284,151.907
C06929=1099.947,88.178,-59.078,176.774,15.284,151.907
C06930=1099.953,88.427,-59.096,176.777,15.284,151.906
C06931=1099.959,88.676,-59.113,176.780,15.285,151.906
C06932=1099.964,88.925,-59.131,176.782,15.285,151.905
C06933=1099.970,89.174,-59.149,176.786,15.285,151.904
C06934=1099.976,89.424,-59.167,176.788,15.286,151.904
C06935=1099.982,89.673,-59.184,176.790,15.286,151.903
C06936=1099.987,89.922,-59.202,176.794,15.286,151.903
C06937=1099.993,90.172,-59.220,176.796,15.286,151.902
C06938=1099.998,90.421,-59.238,176.799,15.287,151.902
C06939=1100.004,90.670,-59.256,176.802,15.287,151.901
C06940=1100.010,90.919,-59.274,176.805,15.287,151.901
C06941=1100.015,91.168,-59.292,176.807,15.287,151.900
C06942=1100.022,91.418,-59.309,176.810,15.288,151.900
C06943=1100.027,91.667,-59.327,176.813,15.288,151.899
C06944=1100.033,91.917,-59.345,176.816,15.288,151.899
C06945=1100.038,92.166,-59.363,176.819,15.288,151.898
C06946=1100.043,92.415,-59.381,176.822,15.289,151.898
C06947=1100.050,92.665,-59.399,176.824,15.289,151.897
C06948=1100.055,92.914,-59.416,176.826,15.289,151.896
C06949=1100.060,93.163,-59.435,176.830,15.289,151.896
C06950=1100.066,93.413,-59.453,176.832,15.289,151.895
C06951=1100.072,93.662,-59.471,176.835,15.290,151.895
C06952=1100.078,93.911,-59.489,176.838,15.290,151.894
C06953=1100.083,94.161,-59.507,176.841,15.290,151.894
C06954=1100.089,94.409,-59.525,176.843,15.290,151.893
C06955=1100.095,94.659,-59.543,176.846,15.291,151.893
C06956=1100.100,94.908,-59.560,176.849,15.291,151.892
C06957=1100.106,95.158,-59.579,176.852,15.291,151.891
C06958=1100.111,95.407,-59.597,176.855,15.291,151.891
C06959=1100.118,95.680,-59.617,176.858,15.292,151.890
C06960=1100.124,95.953,-59.637,176.861,15.292,151.890
C06961=1100.130,96.227,-59.656,176.864,15.292,151.889
C06962=1100.136,96.500,-59.676,176.867,15.292,151.889
C06963=1100.142,96.750,-59.694,176.870,15.293,151.888
C06964=1100.147,96.999,-59.712,176.873,15.293,151.887
C06965=1100.153,97.248,-59.731,176.875,15.293,151.887
C06966=1100.159,97.497,-59.749,176.879,15.293,151.886
C06967=1100.165,97.747,-59.767,176.881,15.293,151.886
C06968=1100.170,97.996,-59.785,176.884,15.293,151.885
C06969=1100.176,98.245,-59.803,176.887,15.293,151.884
C06970=1100.182,98.494,-59.821,176.890,15.294,151.884
C06971=1100.187,98.744,-59.840,176.893,15.293,151.883
C06972=1100.193,98.993,-59.858,176.896,15.294,151.883
C06973=1100.199,99.242,-59.876,176.898,15.294,151.882
C06974=1100.204,99.491,-59.895,176.902,15.294,151.882
C06975=1100.210,99.741,-59.912,176.904,15.294,151.881
C06976=1100.216,99.989,-59.931,176.907,15.295,151.880
C06977=1100.221,100.240,-59.949,176.910,15.294,151.880
C06978=1100.228,100.489,-59.968,176.913,15.295,151.879
C06979=1100.233,100.738,-59.986,176.916,15.295,151.879
C06980=1100.239,100.987,-60.005,176.919,15.295,151.878
C06981=1100.245,101.236,-60.022,176.921,15.295,151.877
C06982=1100.250,101.486,-60.042,176.925,15.296,151.877
C06983=1100.256,101.735,-60.059,176.927,15.295,151.876
C06984=1100.262,101.984,-60.078,176.930,15.296,151.876
C06985=1100.267,102.233,-60.096,176.933,15.296,151.875
C06986=1100.273,102.483,-60.115,176.936,15.296,151.875
C06987=1100.278,102.732,-60.133,176.939,15.296,151.874
C06988=1100.284,102.981,-60.152,176.942,15.297,151.873
C06989=1100.289,103.230,-60.170,176.944,15.296,151.873
C06990=1100.295,103.480,-60.189,176.948,15.297,151.872
C06991=1100.301,103.729,-60.207,176.950,15.297,151.872
C06992=1100.306,103.978,-60.226,176.953,15.297,151.871
C06993=1100.312,104.228,-60.244,176.956,15.297,151.871
C06994=1100.318,104.476,-60.262,176.960,15.297,151.870
C06995=1100.323,104.726,-60.282,176.962,15.297,151.869
C06996=1100.329,104.975,-60.299,176.965,15.297,151.869
C06997=1100.334,105.224,-60.318,176.968,15.297,151.868
C06998=1100.341,105.474,-60.336,176.971,15.298,151.867
C06999=1100.346,105.723,-60.355,176.974,15.298,151.867
C07000=1100.351,105.972,-60.374,176.977,15.298,151.866
C07001=1100.357,106.221,-60.392,176.979,15.298,151.866
C07002=1100.363,106.471,-60.411,176.983,15.298,151.865
C07003=1100.369,106.720,-60.430,176.985,15.298,151.864
C07004=1100.374,106.969,-60.448,176.989,15.298,151.864
C07005=1100.379,107.219,-60.467,176.991,15.298,151.863
C07006=1100.386,107.468,-60.486,176.994,15.299,151.863
C07007=1100.391,107.716,-60.505,176.997,15.298,151.862
C07008=1100.397,107.966,-60.523,177.001,15.299,151.861
C07009=1100.402,108.215,-60.542,177.003,15.298,151.861
C07010=1100.408,108.464,-60.561,177.006,15.299,151.860
C07011=1100.414,108.714,-60.579,177.009,15.299,151.860
C07012=1100.419,108.963,-60.598,177.012,15.299,151.859
C07013=1100.425,109.212,-60.616,177.015,15.299,151.858
C07014=1100.431,109.461,-60.636,177.018,15.299,151.858
C07015=1100.437,109.711,-60.655,177.021,15.298,151.857
C07016=1100.442,109.960,-60.672,177.024,15.299,151.856
C07017=1100.448,110.209,-60.692,177.027,15.299,151.856
C07018=1100.454,110.459,-60.711,177.030,15.299,151.855
C07019=1100.460,110.707,-60.729,177.033,15.299,151.854
C07020=1100.465,110.957,-60.748,177.036,15.299,151.854
C07021=1100.471,111.206,-60.768,177.039,15.299,151.853
C07022=1100.476,111.455,-60.785,177.042,15.299,151.853
C07023=1100.483,111.728,-60.807,177.045,15.299,151.852
C07024=1100.489,112.002,-60.828,177.048,15.299,151.851
C07025=1100.495,112.275,-60.848,177.052,15.299,151.850
C07026=1100.501,112.549,-60.869,177.055,15.299,151.850
C07027=1100.507,112.798,-60.888,177.058,15.299,151.849
C07028=1100.513,113.048,-60.907,177.061,15.299,151.849
C07029=1100.518,113.296,-60.926,177.064,15.299,151.848
C07030=1100.524,113.546,-60.945,177.067,15.299,151.847
C07031=1100.530,113.795,-60.964,177.070,15.299,151.847
C07032=1100.535,114.044,-60.982,177.073,15.299,151.846
C07033=1100.541,114.293,-61.002,177.076,15.299,151.845
C07034=1100.547,114.542,-61.021,177.079,15.300,151.845
C07035=1100.553,114.792,-61.040,177.082,15.299,151.844
C07036=1100.558,115.041,-61.059,177.085,15.299,151.843
C07037=1100.563,115.290,-61.078,177.088,15.299,151.843
C07038=1100.569,115.539,-61.098,177.091,15.299,151.842
C07039=1100.575,115.789,-61.117,177.094,15.299,151.842
C07040=1100.580,116.038,-61.136,177.097,15.299,151.841
C07041=1100.585,116.287,-61.155,177.100,15.299,151.840
C07042=1100.591,116.537,-61.174,177.103,15.300,151.840
C07043=1100.596,116.785,-61.193,177.106,15.299,151.839
C07044=1100.602,117.035,-61.212,177.109,15.299,151.838
C07045=1100.608,117.284,-61.232,177.113,15.300,151.838
C07046=1100.613,117.534,-61.251,177.115,15.299,151.837
C07047=1100.618,117.782,-61.270,177.118,15.300,151.836
C07048=1100.624,118.032,-61.289,177.121,15.299,151.836
C07049=1100.630,118.281,-61.309,177.124,15.300,151.835
C07050=1100.636,118.530,-61.328,177.127,15.299,151.834
C07051=1100.641,118.779,-61.347,177.131,15.300,151.834
C07052=1100.647,119.028,-61.366,177.133,15.299,151.833
C07053=1100.652,119.278,-61.385,177.137,15.300,151.832
C07054=1100.658,119.527,-61.405,177.139,15.299,151.832
C07055=1100.664,119.776,-61.425,177.143,15.300,151.831
C07056=1100.670,120.025,-61.444,177.145,15.299,151.830
C07057=1100.675,120.274,-61.463,177.149,15.299,151.830
C07058=1100.680,120.523,-61.482,177.152,15.299,151.829
C07059=1100.686,120.773,-61.501,177.155,15.299,151.828
C07060=1100.692,121.022,-61.521,177.158,15.299,151.828
C07061=1100.698,121.271,-61.540,177.161,15.299,151.827
C07062=1100.703,121.521,-61.560,177.164,15.299,151.826
C07063=1100.708,121.769,-61.579,177.167,15.299,151.826
C07064=1100.714,122.018,-61.599,177.171,15.299,151.825
C07065=1100.720,122.267,-61.618,177.173,15.299,151.824
C07066=1100.726,122.517,-61.637,177.177,15.299,151.824
C07067=1100.732,122.766,-61.657,177.179,15.299,151.823
C07068=1100.738,123.015,-61.676,177.183,15.299,151.822
C07069=1100.743,123.265,-61.695,177.186,15.298,151.822
C07070=1100.748,123.513,-61.716,177.189,15.298,151.821
C07071=1100.754,123.762,-61.735,177.192,15.298,151.820
C07072=1100.759,124.012,-61.754,177.195,15.298,151.820
C07073=1100.765,124.261,-61.774,177.198,15.298,151.819
C07074=1100.771,124.510,-61.793,177.202,15.298,151.818
C07075=1100.777,124.760,-61.813,177.205,15.298,151.817
C07076=1100.783,125.008,-61.833,177.208,15.298,151.817
C07077=1100.788,125.258,-61.852,177.211,15.298,151.816
C07078=1100.794,125.507,-61.872,177.214,15.297,151.815
C07079=1100.799,125.756,-61.892,177.218,15.297,151.815
C07080=1100.805,126.006,-61.911,177.220,15.297,151.814
C07081=1100.811,126.255,-61.931,177.224,15.297,151.813
C07082=1100.817,126.504,-61.950,177.226,15.297,151.813
C07083=1100.823,126.753,-61.970,177.230,15.297,151.812
C07084=1100.828,127.002,-61.989,177.233,15.296,151.811
C07085=1100.834,127.250,-62.009,177.236,15.297,151.811
C07086=1100.839,127.500,-62.029,177.239,15.296,151.810
C07087=1100.846,127.774,-62.050,177.242,15.296,151.809
C07088=1100.852,128.047,-62.072,177.246,15.296,151.808
C07089=1100.858,128.320,-62.094,177.250,15.296,151.807
C07090=1100.864,128.593,-62.115,177.253,15.296,151.807
C07091=1100.870,128.843,-62.135,177.256,15.295,151.806
C07092=1100.876,129.091,-62.155,177.260,15.295,151.805
C07093=1100.882,129.340,-62.175,177.263,15.295,151.805
C07094=1100.887,129.590,-62.194,177.266,15.295,151.804
C07095=1100.893,129.840,-62.215,177.269,15.295,151.803
C07096=1100.899,130.089,-62.234,177.272,15.295,151.802
C07097=1100.905,130.338,-62.254,177.275,15.294,151.802
C07098=1100.910,130.587,-62.275,177.279,15.294,151.801
C07099=1100.916,130.836,-62.294,177.282,15.294,151.800
C07100=1100.922,131.085,-62.314,177.285,15.294,151.799
C07101=1100.928,131.334,-62.334,177.289,15.294,151.799
C07102=1100.934,131.583,-62.353,177.291,15.293,151.798
C07103=1100.939,131.833,-62.373,177.295,15.293,151.797
C07104=1100.945,132.081,-62.393,177.298,15.293,151.797
C07105=1100.950,132.331,-62.413,177.301,15.293,151.796
C07106=1100.956,132.580,-62.433,177.304,15.292,151.795
C07107=1100.962,132.829,-62.453,177.308,15.292,151.794
C07108=1100.967,133.078,-62.474,177.311,15.292,151.794
C07109=1100.973,133.327,-62.493,177.314,15.292,151.793
C07110=1100.979,133.576,-62.513,177.317,15.291,151.792
C07111=1100.984,133.825,-62.534,177.321,15.291,151.791
C07112=1100.990,134.074,-62.553,177.324,15.291,151.791
C07113=1100.995,134.324,-62.573,177.327,15.291,151.790
C07114=1101.001,134.573,-62.593,177.331,15.291,151.789
C07115=1101.007,134.822,-62.614,177.333,15.290,151.788
C07116=1101.013,135.071,-62.634,177.337,15.290,151.788
C07117=1101.019,135.320,-62.654,177.340,15.290,151.787
C07118=1101.024,135.570,-62.674,177.343,15.290,151.786
C07119=1101.030,135.819,-62.694,177.346,15.289,151.785
C07120=1101.035,136.068,-62.714,177.350,15.289,151.785
C07121=1101.041,136.316,-62.734,177.353,15.289,151.784
C07122=1101.046,136.566,-62.755,177.356,15.289,151.783
C07123=1101.052,136.814,-62.775,177.360,15.289,151.783
C07124=1101.057,137.064,-62.795,177.362,15.288,151.782
C07125=1101.064,137.314,-62.815,177.366,15.288,151.781
C07126=1101.069,137.563,-62.836,177.369,15.288,151.780
C07127=1101.075,137.812,-62.856,177.372,15.288,151.780
C07128=1101.080,138.061,-62.876,177.376,15.288,151.779
C07129=1101.086,138.310,-62.896,177.379,15.287,151.778
C07130=1101.091,138.559,-62.917,177.383,15.287,151.777
C07131=1101.097,138.807,-62.937,177.385,15.286,151.776
C07132=1101.103,139.057,-62.958,177.389,15.286,151.776
C07133=1101.109,139.306,-62.978,177.392,15.286,151.775
C07134=1101.115,139.555,-62.998,177.395,15.286,151.774
C07135=1101.120,139.804,-63.019,177.398,15.285,151.774
C07136=1101.126,140.053,-63.039,177.402,15.286,151.773
C07137=1101.131,140.302,-63.059,177.406,15.285,151.772
C07138=1101.138,140.552,-63.079,177.408,15.285,151.771
C07139=1101.143,140.801,-63.100,177.412,15.285,151.770
C07140=1101.148,141.050,-63.121,177.415,15.284,151.770
C07141=1101.154,141.299,-63.141,177.418,15.284,151.769
C07142=1101.159,141.548,-63.161,177.421,15.284,151.768
C07143=1101.165,141.797,-63.182,177.425,15.283,151.767
C07144=1101.171,142.047,-63.202,177.429,15.283,151.767
C07145=1101.177,142.295,-63.223,177.431,15.283,151.766
C07146=1101.182,142.544,-63.244,177.435,15.283,151.765
C07147=1101.188,142.793,-63.264,177.438,15.282,151.764
C07148=1101.193,143.042,-63.284,177.442,15.282,151.763
C07149=1101.199,143.291,-63.305,177.445,15.281,151.763
C07150=1101.204,143.541,-63.326,177.448,15.281,151.762
C07151=1101.211,143.814,-63.348,177.452,15.281,151.761
C07152=1101.217,144.088,-63.371,177.456,15.281,151.760
C07153=1101.223,144.360,-63.393,177.459,15.281,151.759
C07154=1101.230,144.634,-63.416,177.463,15.280,151.759
C07155=1101.235,144.883,-63.437,177.466,15.280,151.758
C07156=1101.240,145.132,-63.457,177.470,15.279,151.757
C07157=1101.246,145.381,-63.477,177.473,15.279,151.756
C07158=1101.252,145.630,-63.499,177.476,15.279,151.755
C07159=1101.258,145.879,-63.520,177.480,15.278,151.755
C07160=1101.263,146.128,-63.540,177.483,15.278,151.754
C07161=1101.269,146.376,-63.561,177.486,15.278,151.753
C07162=1101.275,146.626,-63.582,177.490,15.277,151.752
C07163=1101.280,146.875,-63.602,177.493,15.277,151.751
C07164=1101.286,147.124,-63.623,177.496,15.276,151.751
C07165=1101.292,147.374,-63.644,177.500,15.276,151.750
C07166=1101.298,147.623,-63.664,177.503,15.276,151.749
C07167=1101.303,147.872,-63.685,177.507,15.275,151.748
C07168=1101.309,148.121,-63.707,177.510,15.275,151.747
C07169=1101.314,148.370,-63.727,177.513,15.275,151.747
C07170=1101.320,148.619,-63.748,177.517,15.275,151.746
C07171=1101.325,148.868,-63.769,177.520,15.274,151.745
C07172=1101.332,149.117,-63.789,177.524,15.274,151.744
C07173=1101.337,149.366,-63.811,177.527,15.273,151.743
C07174=1101.343,149.615,-63.831,177.530,15.273,151.743
C07175=1101.349,149.865,-63.852,177.534,15.273,151.742
C07176=1101.354,150.113,-63.873,177.537,15.272,151.741
C07177=1101.359,150.362,-63.894,177.541,15.272,151.740
C07178=1101.366,150.611,-63.915,177.544,15.271,151.739
C07179=1101.371,150.861,-63.936,177.547,15.271,151.739
C07180=1101.376,151.109,-63.957,177.550,15.271,151.738
C07181=1101.382,151.359,-63.978,177.554,15.270,151.737
C07182=1101.388,151.607,-63.999,177.558,15.270,151.736
C07183=1101.393,151.856,-64.020,177.561,15.269,151.735
C07184=1101.399,152.106,-64.042,177.564,15.269,151.735
C07185=1101.404,152.355,-64.062,177.567,15.268,151.734
C07186=1101.410,152.603,-64.083,177.571,15.269,151.733
C07187=1101.416,152.853,-64.104,177.575,15.268,151.732
C07188=1101.421,153.102,-64.126,177.578,15.267,151.731
C07189=1101.427,153.351,-64.147,177.582,15.267,151.730
C07190=1101.433,153.600,-64.168,177.585,15.266,151.729
C07191=1101.438,153.848,-64.189,177.588,15.266,151.729
C07192=1101.444,154.098,-64.210,177.592,15.266,151.728
C07193=1101.450,154.347,-64.231,177.595,15.265,151.727
C07194=1101.456,154.596,-64.253,177.599,15.265,151.726
C07195=1101.461,154.845,-64.273,177.602,15.264,151.725
C07196=1101.467,155.094,-64.295,177.605,15.264,151.725
C07197=1101.473,155.343,-64.316,177.609,15.264,151.724
C07198=1101.478,155.592,-64.337,177.612,15.263,151.723
C07199=1101.484,155.841,-64.359,177.616,15.263,151.722
C07200=1101.490,156.090,-64.379,177.619,15.262,151.721
C07201=1101.496,156.339,-64.401,177.623,15.262,151.720
C07202=1101.501,156.588,-64.423,177.627,15.262,151.719
C07203=1101.506,156.837,-64.444,177.630,15.261,151.719
C07204=1101.512,157.087,-64.465,177.633,15.261,151.718
C07205=1101.518,157.335,-64.486,177.636,15.260,151.717
C07206=1101.524,157.584,-64.508,177.640,15.260,151.716
C07207=1101.529,157.833,-64.529,177.644,15.260,151.715
C07208=1101.535,158.083,-64.550,177.647,15.259,151.714
C07209=1101.540,158.331,-64.572,177.651,15.258,151.714
C07210=1101.546,158.581,-64.593,177.654,15.258,151.713
C07211=1101.552,158.829,-64.615,177.658,15.258,151.712
C07212=1101.558,159.078,-64.636,177.661,15.257,151.711
C07213=1101.563,159.328,-64.657,177.665,15.256,151.710
C07214=1101.569,159.577,-64.679,177.668,15.256,151.709
C07215=1101.575,159.849,-64.702,177.672,15.256,151.708
C07216=1101.581,160.123,-64.726,177.675,15.255,151.707
C07217=1101.587,160.395,-64.749,177.679,15.254,151.707
C07218=1101.593,160.668,-64.773,177.683,15.254,151.706
C07219=1101.600,160.918,-64.795,177.687,15.254,151.705
C07220=1101.605,161.166,-64.816,177.690,15.253,151.704
C07221=1101.611,161.416,-64.838,177.694,15.252,151.703
C07222=1101.616,161.664,-64.859,177.698,15.252,151.702
C07223=1101.622,161.913,-64.881,177.701,15.251,151.701
C07224=1101.627,162.162,-64.903,177.705,15.251,151.700
C07225=1101.633,162.411,-64.924,177.708,15.250,151.700
C07226=1101.639,162.660,-64.946,177.711,15.250,151.699
C07227=1101.644,162.909,-64.968,177.715,15.250,151.698
C07228=1101.650,163.158,-64.989,177.718,15.249,151.697
C07229=1101.655,163.407,-65.011,177.722,15.249,151.696
C07230=1101.661,163.656,-65.033,177.726,15.249,151.695
C07231=1101.666,163.905,-65.055,177.729,15.248,151.694
C07232=1101.672,164.154,-65.076,177.733,15.247,151.694
C07233=1101.677,164.403,-65.098,177.736,15.246,151.693
C07234=1101.683,164.652,-65.120,177.740,15.247,151.692
C07235=1101.688,164.901,-65.142,177.743,15.246,151.691
C07236=1101.694,165.150,-65.163,177.747,15.245,151.690
C07237=1101.699,165.399,-65.185,177.750,15.245,151.689
C07238=1101.705,165.648,-65.207,177.754,15.245,151.688
C07239=1101.710,165.897,-65.229,177.757,15.244,151.687
C07240=1101.716,166.146,-65.250,177.761,15.244,151.687
C07241=1101.721,166.395,-65.272,177.764,15.243,151.686
C07242=1101.727,166.644,-65.294,177.768,15.242,151.685
C07243=1101.732,166.893,-65.317,177.772,15.242,151.684
C07244=1101.739,167.142,-65.338,177.775,15.241,151.683
C07245=1101.743,167.391,-65.360,177.779,15.241,151.682
C07246=1101.750,167.640,-65.382,177.783,15.241,151.681
C07247=1101.754,167.889,-65.404,177.786,15.240,151.680
C07248=1101.761,168.138,-65.425,177.790,15.239,151.680
C07249=1101.766,168.387,-65.448,177.793,15.238,151.679
C07250=1101.772,168.635,-65.470,177.796,15.238,151.678
C07251=1101.777,168.885,-65.492,177.800,15.238,151.677
C07252=1101.783,169.134,-65.513,177.803,15.237,151.676
C07253=1101.789,169.382,-65.536,177.807,15.237,151.675
C07254=1101.794,169.632,-65.558,177.811,15.237,151.674
C07255=1101.800,169.880,-65.579,177.814,15.236,151.674
C07256=1101.805,170.130,-65.602,177.818,15.235,151.673
C07257=1101.812,170.379,-65.624,177.821,15.234,151.672
C07258=1101.816,170.627,-65.646,177.825,15.234,151.671
C07259=1101.822,170.877,-65.668,177.829,15.234,151.670
C07260=1101.828,171.125,-65.690,177.832,15.233,151.669
C07261=1101.833,171.374,-65.712,177.836,15.232,151.668
C07262=1101.839,171.623,-65.734,177.840,15.232,151.667
C07263=1101.845,171.872,-65.757,177.843,15.231,151.666
C07264=1101.850,172.121,-65.779,177.847,15.230,151.665
C07265=1101.856,172.370,-65.801,177.851,15.230,151.664
C07266=1101.862,172.619,-65.823,177.854,15.229,151.664
C07267=1101.867,172.869,-65.846,177.858,15.229,151.663
